# B&R Automation Studio project Panasonic_LinkaPowerCP2_A2021055 (part 34)

#### Main.st - Init, cyclic, exit code
```iecst
PROGRAM _INIT
	(* Insert code here *)

END_PROGRAM

PROGRAM _CYCLIC

	//**********************************************************IO modul Wedmuller**********************************************************************//
	//************Karta AB 4.2 8DI**************//
	P4_Etiketovacka.IN.NapajanieTlaciarne_OK := P4_Pracovisko.COM_Weidmuller.AB4_2_8DI.0;
	P4_Vytah.IN.StavRiadeniaDopravVytahu_READY := P4_Pracovisko.COM_Weidmuller.AB4_2_8DI.1;
	P4_Dopravniky.IN.StavRiadPredDopravBunky_READY := P4_Pracovisko.COM_Weidmuller.AB4_2_8DI.2;
	P4_Dopravniky.IN.StavRiadeniaPriecnDoprav_READY := P4_Pracovisko.COM_Weidmuller.AB4_2_8DI.3;
	P4_Dopravniky.IN.StavRiadZadnDopravBunky_READY := P4_Pracovisko.COM_Weidmuller.AB4_2_8DI.4;
	P4_Dopravniky.IN.StavRiadeniaVratnehoDoprav_READY := P4_Pracovisko.COM_Weidmuller.AB4_2_8DI.5;
	P4_Vytah.IN.TeplotaMotoraDopravVytahu_OK := P4_Pracovisko.COM_Weidmuller.AB4_2_8DI.6;
	P4_Dopravniky.IN.TeplotaMotoraPredDopravBunky_OK := P4_Pracovisko.COM_Weidmuller.AB4_2_8DI.7;

	//************Karta AB 4.3 8DI**************//
	P4_Dopravniky.IN.TeplotaMotoraPriecnDoprav_OK := P4_Pracovisko.COM_Weidmuller.AB4_3_8DI.0;
	P4_Dopravniky.IN.TeplotaMotoraZadnDopravBunky_OK := P4_Pracovisko.COM_Weidmuller.AB4_3_8DI.1;
	P4_Dopravniky.IN.TeplotaMotoraVratnehoDoprav_OK :=  P4_Pracovisko.COM_Weidmuller.AB4_3_8DI.2;
	P4_Pracovisko.COM_Weidmuller.AB4_3_8DI.3;
	P4_Pracovisko.COM_Weidmuller.AB4_3_8DI.4;
	P4_Pracovisko.COM_Weidmuller.AB4_3_8DI.5;
	Safety.IN.Linka_SV_ZonaCS := P4_Pracovisko.COM_Weidmuller.AB4_3_8DI.6;
	Safety.IN.P4_SV_ZonaBunky := P4_Pracovisko.COM_Weidmuller.AB4_3_8DI.7;

	//************Karta AB 4.4 8DI**************//
	Safety.IN.P4_SV_ZonaVytahu := P4_Pracovisko.COM_Weidmuller.AB4_4_8DI.0;
	Safety.IN.P4_SV_PrivodVzduchu_CH1 := P4_Pracovisko.COM_Weidmuller.AB4_4_8DI.1;
	Safety.IN.P4_SV_PrivodVzduchu_CH2 := P4_Pracovisko.COM_Weidmuller.AB4_4_8DI.2;
	P4_Pracovisko.IN.TlakVzduchu_OK := P4_Pracovisko.COM_Weidmuller.AB4_4_8DI.3;
	P4_Pracovisko.COM_Weidmuller.AB4_4_8DI.4;
	P4_Pracovisko.COM_Weidmuller.AB4_4_8DI.5;
	P4_Pracovisko.COM_Weidmuller.AB4_4_8DI.6;
	P4_Pracovisko.COM_Weidmuller.AB4_4_8DI.7;

	//************Karta AB 4.5 8DO**************//
	P4_Pracovisko.COM_Weidmuller.AB4_5_8DO.0 := P4_Pracovisko.OUT.Majak_ZeleneSvetlo_ON;
	P4_Pracovisko.COM_Weidmuller.AB4_5_8DO.1 := P4_Pracovisko.OUT.Majak_OranzoveSvetlo_ON;
	P4_Pracovisko.COM_Weidmuller.AB4_5_8DO.2 := P4_Pracovisko.OUT.Majak_CerveneSvetlo_ON;
	P4_Pracovisko.COM_Weidmuller.AB4_5_8DO.3 := P4_Pracovisko.OUT.Majak_Hukacka_ON;
	P4_Pracovisko.COM_Weidmuller.AB4_5_8DO.4;
	P4_Pracovisko.COM_Weidmuller.AB4_5_8DO.5;
	P4_Pracovisko.COM_Weidmuller.AB4_5_8DO.6 := P4_Vytah.OUT.OsvetlenieVytahu_ON;
	P4_Pracovisko.COM_Weidmuller.AB4_5_8DO.7 := P4_Pracovisko.OUT.OsvetlenieBunky_ON;

	//************Karta AB 4.6 8DO**************//
	P4_Pracovisko.COM_Weidmuller.AB4_6_8DO.0 := P4_Pracovisko.OUT.Osvetlenie_CAM15_ON;
	P4_Pracovisko.COM_Weidmuller.AB4_6_8DO.1 := P4_Vytah.OUT.DopravnikChod_VZAD;
	P4_Pracovisko.COM_Weidmuller.AB4_6_8DO.2 := P4_Vytah.OUT.DopravnikChod_VPRED;
	P4_Pracovisko.COM_Weidmuller.AB4_6_8DO.3 := P4_Dopravniky.OUT.PrednyDopravnikBunky_ON;
	P4_Pracovisko.COM_Weidmuller.AB4_6_8DO.4 := P4_Dopravniky.OUT.PriecnyDopravnik_VPRED;
	P4_Pracovisko.COM_Weidmuller.AB4_6_8DO.5 := P4_Dopravniky.OUT.ZadnyDopravnikBunky_ON;
	P4_Pracovisko.COM_Weidmuller.AB4_6_8DO.6 := P4_Dopravniky.OUT.VratnyDopravnik_ON;
	P4_Pracovisko.COM_Weidmuller.AB4_6_8DO.7 := Safety.OUT.Linka_ResetCS;

	//************Karta AB 4.8 8DO**************//
	P4_Pracovisko.COM_Weidmuller.AB4_8_8DO.0:= Safety.OUT.P4_ResetZonyBunky;
	P4_Pracovisko.COM_Weidmuller.AB4_8_8DO.1:= Safety.OUT.P4_ResetZonyVytahu;
	P4_Pracovisko.COM_Weidmuller.AB4_8_8DO.2;
	P4_Pracovisko.COM_Weidmuller.AB4_8_8DO.3;
	P4_Pracovisko.COM_Weidmuller.AB4_8_8DO.4;
	P4_Pracovisko.COM_Weidmuller.AB4_8_8DO.5;
	P4_Pracovisko.COM_Weidmuller.AB4_8_8DO.6;
	P4_Pracovisko.COM_Weidmuller.AB4_8_8DO.7;

	//**************************************************************IO modul Festo**********************************************************************************//

	//**********Modul DM 4.1 4DI4DO**************//
	//Inputs//
	P4_Pracovisko.IN.PredneDvere_PritomnostAdaptera := P4_Pracovisko.COM_Festo.DM4_1_4DI[0];
	P4_Pracovisko.IN.ZadneDvere_PritomnostAdaptera := P4_Pracovisko.COM_Festo.DM4_1_4DI[1];
	P4_ZdvizkaZaFunkcTestA.IN.TlmicPaletky_ZASUNUTY := P4_Pracovisko.COM_Festo.DM4_1_4DI[2];
	P4_Vytah.IN.PrechodDopravnika := P4_Pracovisko.COM_Festo.DM4_1_4DI[3];

	//Outputs//
	P4_Pracovisko.COM_Festo.DM4_1_4DO[0] := P4_Pracovisko.OUT.PredneDvere_ZAMKNI;
	P4_Pracovisko.COM_Festo.DM4_1_4DO[1] := P4_Pracovisko.OUT.ZadneDvere_ZAMKNI;
	P4_Pracovisko.COM_Festo.DM4_1_4DO[2];
	P4_Pracovisko.COM_Festo.DM4_1_4DO[3];

	//***********Modul DI 4.1 8DI****************//
	P4_FunkcnyTestA.IN.TypSpodnychKontaktov_5F_5H:= P4_Pracovisko.COM_Festo.DI4_1_8DI[0];
	P4_FunkcnyTestA.IN.TypSpodnychKontaktov_4F:= P4_Pracovisko.COM_Festo.DI4_1_8DI[1];
	P4_FunkcnyTestB.IN.TypSpodnychKontaktov_5F_5H:= P4_Pracovisko.COM_Festo.DI4_1_8DI[2];
	P4_FunkcnyTestB.IN.TypSpodnychKontaktov_4F:= P4_Pracovisko.COM_Festo.DI4_1_8DI[3];
	P4_Etiketovacka.IN.Centrovanie_ZASUNUTE := P4_Pracovisko.COM_Festo.DI4_1_8DI[4];
	P4_Etiketovacka.IN.Centrovanie_VYSUNUTE := P4_Pracovisko.COM_Festo.DI4_1_8DI[5];
	P4_SpodnyStoper.IN.ZaplnenieDopravnika := P4_Pracovisko.COM_Festo.DI4_1_8DI[6];
	P4_SpodnyStoper.IN.PritomnostPaletky := P4_Pracovisko.COM_Festo.DI4_1_8DI[7];

	//***********Modul DI 4.2 8DI****************//
	P4_Etiketovacka.IN.Aplikator_OtocenyVPRED := P4_Pracovisko.COM_Festo.DI4_2_8DI[0];
	P4_Etiketovacka.IN.Aplikator_OtocenyVZAD := P4_Pracovisko.COM_Festo.DI4_2_8DI[1];
	P4_Etiketovacka.IN.Aplikator_ZASUNUTY := P4_Pracovisko.COM_Festo.DI4_2_8DI[2];
	P4_Etiketovacka.IN.Aplikator_VYSUNUTY := P4_Pracovisko.COM_Festo.DI4_2_8DI[3];
	P4_Etiketovacka.IN.PritlakPowerCP_ZASUNUTY := P4_Pracovisko.COM_Festo.DI4_2_8DI[4];
	P4_Etiketovacka.IN.PritlakPowerCP_VYSUNUTY_45F := P4_Pracovisko.COM_Festo.DI4_2_8DI[5];
	P4_Etiketovacka.IN.PrisavanieEtikety_Vakum_OK := P4_Pracovisko.COM_Festo.DI4_2_8DI[6];
	P4_Etiketovacka.IN.PritlakPowerCP_VYSUNUTY_5H := P4_Pracovisko.COM_Festo.DI4_2_8DI[7];

	//***********Modul DI 4.3 8DI****************//
	P4_FunkcnyTestA.IN.HorneKontakty_VYSUNUTE := P4_Pracovisko.COM_Festo.DI4_3_8DI[0];
	P4_FunkcnyTestA.IN.HorneKontakty_ZASUNUTE := P4_Pracovisko.COM_Festo.DI4_3_8DI[1];
	P4_FunkcnyTestA.IN.Centrovanie_ZASUNUTE := P4_Pracovisko.COM_Festo.DI4_3_8DI[2];
	P4_FunkcnyTestA.IN.Centrovanie_VYSUNUTE := P4_Pracovisko.COM_Festo.DI4_3_8DI[3];
	P4_FunkcnyTestA.IN.SpodneKontakty_ZASUNUTE := P4_Pracovisko.COM_Festo.DI4_3_8DI[4];
	P4_FunkcnyTestA.IN.SpodneKontakty_VYSUNUTE := P4_Pracovisko.COM_Festo.DI4_3_8DI[5];
	P4_Pracovisko.COM_Festo.DI4_3_8DI[6];
	P4_Pracovisko.COM_Festo.DI4_3_8DI[7];

	//***********Modul DI 4.4 8DI****************//
	P4_FunkcnyTestB.IN.HorneKontakty_VYSUNUTE := P4_Pracovisko.COM_Festo.DI4_4_8DI[0];
	P4_FunkcnyTestB.IN.HorneKontakty_ZASUNUTE := P4_Pracovisko.COM_Festo.DI4_4_8DI[1];
	P4_FunkcnyTestB.IN.Centrovanie_ZASUNUTE := P4_Pracovisko.COM_Festo.DI4_4_8DI[2];
	P4_FunkcnyTestB.IN.Centrovanie_VYSUNUTE := P4_Pracovisko.COM_Festo.DI4_4_8DI[3];
	P4_FunkcnyTestB.IN.SpodneKontakty_ZASUNUTE := P4_Pracovisko.COM_Festo.DI4_4_8DI[4];
	P4_FunkcnyTestB.IN.SpodneKontakty_VYSUNUTE := P4_Pracovisko.COM_Festo.DI4_4_8DI[5];
	P4_Pracovisko.COM_Festo.DI4_4_8DI[6];
	P4_Pracovisko.COM_Festo.DI4_4_8DI[7];

	//***********Modul DI 4.5 8DI****************//
	P4_ZdvizkaZaFunkcTestA.IN.Zdvizka_HornaPoloha := P4_Pracovisko.COM_Festo.DI4_5_8DI[0];
	P4_ZdvizkaZaFunkcTestA.IN.Zdvizka_SpodnaPoloha := P4_Pracovisko.COM_Festo.DI4_5_8DI[1];
	P4_ZdvizkaZaFunkcTestA.IN.PoziciaPaletky_OK := P4_Pracovisko.COM_Festo.DI4_5_8DI[2];
	P4_ZdvizkaZaFunkcTestA.IN.Zdvizka_StrednaPoloha := P4_Pracovisko.COM_Festo.DI4_5_8DI[3];
	P4_ZdvizkaZaFunkcTestB.IN.PritomnostPaletky := P4_Pracovisko.COM_Festo.DI4_5_8DI[4];
	P4_ZdvizkaZaFunkcTestA.IN.PritomnostPaletky := P4_Pracovisko.COM_Festo.DI4_5_8DI[5];
	P4_ZdvizkaZaFunkcTestB.IN.Zdvizka_StrednaPoloha := P4_Pracovisko.COM_Festo.DI4_5_8DI[6];
	P4_ZdvizkaZaFunkcTestB.IN.Zdvizka_HornaPoloha := P4_Pracovisko.COM_Festo.DI4_5_8DI[7];

	//********Modul DS 4.1 IO link Port 0 - RFID snímač paletky funkčný test A**************//
	//Inputs//
	P4_FunkcnyTestA.RFID_hlava.Mapping_IN[0]:= P4_Pracovisko.COM_Festo.DS4_1_Port0_IN[0];
	P4_FunkcnyTestA.RFID_hlava.Mapping_IN[1]:= P4_Pracovisko.COM_Festo.DS4_1_Port0_IN[1];
	P4_FunkcnyTestA.RFID_hlava.Mapping_IN[2]:= P4_Pracovisko.COM_Festo.DS4_1_Port0_IN[2];
	P4_FunkcnyTestA.RFID_hlava.Mapping_IN[3]:= P4_Pracovisko.COM_Festo.DS4_1_Port0_IN[3];
	P4_FunkcnyTestA.RFID_hlava.Mapping_IN[4]:= P4_Pracovisko.COM_Festo.DS4_1_Port0_IN[4];
	P4_FunkcnyTestA.RFID_hlava.Mapping_IN[5]:= P4_Pracovisko.COM_Festo.DS4_1_Port0_IN[5];
	P4_FunkcnyTestA.RFID_hlava.Mapping_IN[6]:= P4_Pracovisko.COM_Festo.DS4_1_Port0_IN[6];
	P4_FunkcnyTestA.RFID_hlava.Mapping_IN[7]:= P4_Pracovisko.COM_Festo.DS4_1_Port0_IN[7];

	//Outputs//
	P4_Pracovisko.COM_Festo.DS4_1_Port0_OUT[0]:= P4_FunkcnyTestA.RFID_hlava.Mapping_OUT[0];
	P4_Pracovisko.COM_Festo.DS4_1_Port0_OUT[1]:= P4_FunkcnyTestA.RFID_hlava.Mapping_OUT[1];
	P4_Pracovisko.COM_Festo.DS4_1_Port0_OUT[2]:= P4_FunkcnyTestA.RFID_hlava.Mapping_OUT[2];
	P4_Pracovisko.COM_Festo.DS4_1_Port0_OUT[3]:= P4_FunkcnyTestA.RFID_hlava.Mapping_OUT[3];
	P4_Pracovisko.COM_Festo.DS4_1_Port0_OUT[4]:= P4_FunkcnyTestA.RFID_hlava.Mapping_OUT[4];
	P4_Pracovisko.COM_Festo.DS4_1_Port0_OUT[5]:= P4_FunkcnyTestA.RFID_hlava.Mapping_OUT[5];
	P4_Pracovisko.COM_Festo.DS4_1_Port0_OUT[6]:= P4_FunkcnyTestA.RFID_hlava.Mapping_OUT[6];
	P4_Pracovisko.COM_Festo.DS4_1_Port0_OUT[7]:= P4_FunkcnyTestA.RFID_hlava.Mapping_OUT[7];

	//********Modul DS 4.1 IO link Port 1 - RFID snímač paletky funkčný test B**************//
	//Inputs//
	P4_FunkcnyTestB.RFID_hlava.Mapping_IN[0]:= P4_Pracovisko.COM_Festo.DS4_1_Port1_IN[0];
	P4_FunkcnyTestB.RFID_hlava.Mapping_IN[1]:= P4_Pracovisko.COM_Festo.DS4_1_Port1_IN[1];
	P4_FunkcnyTestB.RFID_hlava.Mapping_IN[2]:= P4_Pracovisko.COM_Festo.DS4_1_Port1_IN[2];
	P4_FunkcnyTestB.RFID_hlava.Mapping_IN[3]:= P4_Pracovisko.COM_Festo.DS4_1_Port1_IN[3];
	P4_FunkcnyTestB.RFID_hlava.Mapping_IN[4]:= P4_Pracovisko.COM_Festo.DS4_1_Port1_IN[4];
	P4_FunkcnyTestB.RFID_hlava.Mapping_IN[5]:= P4_Pracovisko.COM_Festo.DS4_1_Port1_IN[5];
	P4_FunkcnyTestB.RFID_hlava.Mapping_IN[6]:= P4_Pracovisko.COM_Festo.DS4_1_Port1_IN[6];
	P4_FunkcnyTestB.RFID_hlava.Mapping_IN[7]:= P4_Pracovisko.COM_Festo.DS4_1_Port1_IN[7];

	//Outputs//
	P4_Pracovisko.COM_Festo.DS4_1_Port1_OUT[0]:= P4_FunkcnyTestB.RFID_hlava.Mapping_OUT[0];
	P4_Pracovisko.COM_Festo.DS4_1_Port1_OUT[1]:= P4_FunkcnyTestB.RFID_hlava.Mapping_OUT[1];
	P4_Pracovisko.COM_Festo.DS4_1_Port1_OUT[2]:= P4_FunkcnyTestB.RFID_hlava.Mapping_OUT[2];
	P4_Pracovisko.COM_Festo.DS4_1_Port1_OUT[3]:= P4_FunkcnyTestB.RFID_hlava.Mapping_OUT[3];
	P4_Pracovisko.COM_Festo.DS4_1_Port1_OUT[4]:= P4_FunkcnyTestB.RFID_hlava.Mapping_OUT[4];
	P4_Pracovisko.COM_Festo.DS4_1_Port1_OUT[5]:= P4_FunkcnyTestB.RFID_hlava.Mapping_OUT[5];
	P4_Pracovisko.COM_Festo.DS4_1_Port1_OUT[6]:= P4_FunkcnyTestB.RFID_hlava.Mapping_OUT[6];
	P4_Pracovisko.COM_Festo.DS4_1_Port1_OUT[7]:= P4_FunkcnyTestB.RFID_hlava.Mapping_OUT[7];

	//********Modul DS 4.1 IO link Port 2 - RFID snímač paletky etiketovanie**************//
	//Inputs//
	P4_Etiketovacka.RFID_hlava.Mapping_IN[0]:= P4_Pracovisko.COM_Festo.DS4_1_Port2_IN[0];
	P4_Etiketovacka.RFID_hlava.Mapping_IN[1]:= P4_Pracovisko.COM_Festo.DS4_1_Port2_IN[1];
	P4_Etiketovacka.RFID_hlava.Mapping_IN[2]:= P4_Pracovisko.COM_Festo.DS4_1_Port2_IN[2];
	P4_Etiketovacka.RFID_hlava.Mapping_IN[3]:= P4_Pracovisko.COM_Festo.DS4_1_Port2_IN[3];
	P4_Etiketovacka.RFID_hlava.Mapping_IN[4]:= P4_Pracovisko.COM_Festo.DS4_1_Port2_IN[4];
	P4_Etiketovacka.RFID_hlava.Mapping_IN[5]:= P4_Pracovisko.COM_Festo.DS4_1_Port2_IN[5];
	P4_Etiketovacka.RFID_hlava.Mapping_IN[6]:= P4_Pracovisko.COM_Festo.DS4_1_Port2_IN[6];
	P4_Etiketovacka.RFID_hlava.Mapping_IN[7]:= P4_Pracovisko.COM_Festo.DS4_1_Port2_IN[7];

	//Outputs//
	P4_Pracovisko.COM_Festo.DS4_1_Port2_OUT[0]:= P4_Etiketovacka.RFID_hlava.Mapping_OUT[0];
	P4_Pracovisko.COM_Festo.DS4_1_Port2_OUT[1]:= P4_Etiketovacka.RFID_hlava.Mapping_OUT[1];
	P4_Pracovisko.COM_Festo.DS4_1_Port2_OUT[2]:= P4_Etiketovacka.RFID_hlava.Mapping_OUT[2];
	P4_Pracovisko.COM_Festo.DS4_1_Port2_OUT[3]:= P4_Etiketovacka.RFID_hlava.Mapping_OUT[3];
	P4_Pracovisko.COM_Festo.DS4_1_Port2_OUT[4]:= P4_Etiketovacka.RFID_hlava.Mapping_OUT[4];
	P4_Pracovisko.COM_Festo.DS4_1_Port2_OUT[5]:= P4_Etiketovacka.RFID_hlava.Mapping_OUT[5];
	P4_Pracovisko.COM_Festo.DS4_1_Port2_OUT[6]:= P4_Etiketovacka.RFID_hlava.Mapping_OUT[6];
	P4_Pracovisko.COM_Festo.DS4_1_Port2_OUT[7]:= P4_Etiketovacka.RFID_hlava.Mapping_OUT[7];

	//*************Modul DS 4.2 IO link Port 0 - Banner*********************//
	//Inputs//
	P4_Vytah.Banner.Mapping_IN[0]:= P4_Pracovisko.COM_Festo.DS4_2_Port0_IN[0];
	P4_Vytah.Banner.Mapping_IN[1]:= P4_Pracovisko.COM_Festo.DS4_2_Port0_IN[1];
	P4_Vytah.Banner.Mapping_IN[2]:= P4_Pracovisko.COM_Festo.DS4_2_Port0_IN[2];
	P4_Vytah.Banner.Mapping_IN[3]:= P4_Pracovisko.COM_Festo.DS4_2_Port0_IN[3];
	P4_Vytah.Banner.Mapping_IN[4]:= P4_Pracovisko.COM_Festo.DS4_2_Port0_IN[4];
	P4_Vytah.Banner.Mapping_IN[5]:= P4_Pracovisko.COM_Festo.DS4_2_Port0_IN[5];
	P4_Vytah.Banner.Mapping_IN[6]:= P4_Pracovisko.COM_Festo.DS4_2_Port0_IN[6];
	P4_Vytah.Banner.Mapping_IN[7]:= P4_Pracovisko.COM_Festo.DS4_2_Port0_IN[7];
	P4_Vytah.Banner.Mapping_IN[8]:= P4_Pracovisko.COM_Festo.DS4_2_Port0_IN[8];
	P4_Vytah.Banner.Mapping_IN[9]:= P4_Pracovisko.COM_Festo.DS4_2_Port0_IN[9];
	P4_Vytah.Banner.Mapping_IN[10]:= P4_Pracovisko.COM_Festo.DS4_2_Port0_IN[10];
	P4_Vytah.Banner.Mapping_IN[11]:= P4_Pracovisko.COM_Festo.DS4_2_Port0_IN[11];
	P4_Vytah.Banner.Mapping_IN[12]:= P4_Pracovisko.COM_Festo.DS4_2_Port0_IN[12];
	P4_Vytah.Banner.Mapping_IN[13]:= P4_Pracovisko.COM_Festo.DS4_2_Port0_IN[13];
	P4_Vytah.Banner.Mapping_IN[14]:= P4_Pracovisko.COM_Festo.DS4_2_Port0_IN[14];
	P4_Vytah.Banner.Mapping_IN[15]:= P4_Pracovisko.COM_Festo.DS4_2_Port0_IN[15];

	//Outputs//
	P4_Pracovisko.COM_Festo.DS4_2_Port0_OUT[0]:= P4_Vytah.Banner.Mapping_OUT[0];
	P4_Pracovisko.COM_Festo.DS4_2_Port0_OUT[1]:= P4_Vytah.Banner.Mapping_OUT[1];
	P4_Pracovisko.COM_Festo.DS4_2_Port0_OUT[2]:= P4_Vytah.Banner.Mapping_OUT[2];
	P4_Pracovisko.COM_Festo.DS4_2_Port0_OUT[3]:= P4_Vytah.Banner.Mapping_OUT[3];
	P4_Pracovisko.COM_Festo.DS4_2_Port0_OUT[4]:= P4_Vytah.Banner.Mapping_OUT[4];
	P4_Pracovisko.COM_Festo.DS4_2_Port0_OUT[5]:= P4_Vytah.Banner.Mapping_OUT[5];
	P4_Pracovisko.COM_Festo.DS4_2_Port0_OUT[6]:= P4_Vytah.Banner.Mapping_OUT[6];
	P4_Pracovisko.COM_Festo.DS4_2_Port0_OUT[7]:= P4_Vytah.Banner.Mapping_OUT[7];
	P4_Pracovisko.COM_Festo.DS4_2_Port0_OUT[8]:= P4_Vytah.Banner.Mapping_OUT[8];
	P4_Pracovisko.COM_Festo.DS4_2_Port0_OUT[9]:= P4_Vytah.Banner.Mapping_OUT[9];
	P4_Pracovisko.COM_Festo.DS4_2_Port0_OUT[10]:= P4_Vytah.Banner.Mapping_OUT[10];
	P4_Pracovisko.COM_Festo.DS4_2_Port0_OUT[11]:= P4_Vytah.Banner.Mapping_OUT[11];
	P4_Pracovisko.COM_Festo.DS4_2_Port0_OUT[12]:= P4_Vytah.Banner.Mapping_OUT[12];
	P4_Pracovisko.COM_Festo.DS4_2_Port0_OUT[13]:= P4_Vytah.Banner.Mapping_OUT[13];
	P4_Pracovisko.COM_Festo.DS4_2_Port0_OUT[14]:= P4_Vytah.Banner.Mapping_OUT[14];
	P4_Pracovisko.COM_Festo.DS4_2_Port0_OUT[15]:= P4_Vytah.Banner.Mapping_OUT[15];

	//********Modul DS 4.2 IO link Port 1 - RFID snímač paletky výstupný výťah**************//
	//Inputs//
	P4_Vytah.RFID_hlava.Mapping_IN[0]:= P4_Pracovisko.COM_Festo.DS4_2_Port1_IN[0];
	P4_Vytah.RFID_hlava.Mapping_IN[1]:= P4_Pracovisko.COM_Festo.DS4_2_Port1_IN[1];
	P4_Vytah.RFID_hlava.Mapping_IN[2]:= P4_Pracovisko.COM_Festo.DS4_2_Port1_IN[2];
	P4_Vytah.RFID_hlava.Mapping_IN[3]:= P4_Pracovisko.COM_Festo.DS4_2_Port1_IN[3];
	P4_Vytah.RFID_hlava.Mapping_IN[4]:= P4_Pracovisko.COM_Festo.DS4_2_Port1_IN[4];
	P4_Vytah.RFID_hlava.Mapping_IN[5]:= P4_Pracovisko.COM_Festo.DS4_2_Port1_IN[5];
	P4_Vytah.RFID_hlava.Mapping_IN[6]:= P4_Pracovisko.COM_Festo.DS4_2_Port1_IN[6];
	P4_Vytah.RFID_hlava.Mapping_IN[7]:= P4_Pracovisko.COM_Festo.DS4_2_Port1_IN[7];

	//Outputs//
	P4_Pracovisko.COM_Festo.DS4_2_Port1_OUT[0]:= P4_Vytah.RFID_hlava.Mapping_OUT[0];
	P4_Pracovisko.COM_Festo.DS4_2_Port1_OUT[1]:= P4_Vytah.RFID_hlava.Mapping_OUT[1];
	P4_Pracovisko.COM_Festo.DS4_2_Port1_OUT[2]:= P4_Vytah.RFID_hlava.Mapping_OUT[2];
	P4_Pracovisko.COM_Festo.DS4_2_Port1_OUT[3]:= P4_Vytah.RFID_hlava.Mapping_OUT[3];
	P4_Pracovisko.COM_Festo.DS4_2_Port1_OUT[4]:= P4_Vytah.RFID_hlava.Mapping_OUT[4];
	P4_Pracovisko.COM_Festo.DS4_2_Port1_OUT[5]:= P4_Vytah.RFID_hlava.Mapping_OUT[5];
	P4_Pracovisko.COM_Festo.DS4_2_Port1_OUT[6]:= P4_Vytah.RFID_hlava.Mapping_OUT[6];
	P4_Pracovisko.COM_Festo.DS4_2_Port1_OUT[7]:= P4_Vytah.RFID_hlava.Mapping_OUT[7];

	//************************************Ventilový terminál*******************************************//
	//0-7
	P4_Pracovisko.COM_VentilovyTerminal[0].0 := P4_Etiketovacka.OUT.PrisavanieEtikety_ON;
	P4_Pracovisko.COM_VentilovyTerminal[0].1 := P4_Etiketovacka.OUT.PrisavanieEtikety_OFF;
	P4_Pracovisko.COM_VentilovyTerminal[0].2 := P4_FunkcnyTestA.OUT.ZasunStoper;
	P4_Pracovisko.COM_VentilovyTerminal[0].3 := P4_FunkcnyTestB.OUT.ZasunStoper;
	P4_Pracovisko.COM_VentilovyTerminal[0].4 := P4_ZdvizkaZaFunkcTestA.OUT.Zdvizku_VYSUN;
	P4_Pracovisko.COM_VentilovyTerminal[0].5 := P4_ZdvizkaZaFunkcTestA.OUT.Zdvizku_ZASUN;
	P4_Pracovisko.COM_VentilovyTerminal[0].6 := P4_ZdvizkaZaFunkcTestA.OUT.TlmicPaletky_VYSUN;
	P4_Pracovisko.COM_VentilovyTerminal[0].7 := P4_ZdvizkaZaFunkcTestA.OUT.TlmicPaletky_ZASUN;

	//8-15
	P4_Pracovisko.COM_VentilovyTerminal[1].0 := P4_ZdvizkaZaFunkcTestB.OUT.Zdvizku_VYSUN;
	P4_Pracovisko.COM_VentilovyTerminal[1].1 := P4_Pracovisko.OUT.ZdvizkyPneuZamok_ODOMKNI;
	P4_Pracovisko.COM_VentilovyTerminal[1].2 := P4_ZdvizkaZaFunkcTestB.OUT.TlmicPaletky_VYSUN;
	P4_Pracovisko.COM_VentilovyTerminal[1].3 := P4_Etiketovacka.OUT.ZasunStoper;
	P4_Pracovisko.COM_VentilovyTerminal[1].4 := P4_SpodnyStoper.OUT.ZasunStoper;
	P4_Pracovisko.COM_VentilovyTerminal[1].5;
	P4_Pracovisko.COM_VentilovyTerminal[1].6 := P4_FunkcnyTestA.OUT.PritlakPowerCP_VYSUN;
	P4_Pracovisko.COM_VentilovyTerminal[1].7;

	//16-23
	P4_Pracovisko.COM_VentilovyTerminal[2].0 := P4_FunkcnyTestB.OUT.PritlakPowerCP_VYSUN;
	P4_Pracovisko.COM_VentilovyTerminal[2].1;
	P4_Pracovisko.COM_VentilovyTerminal[2].2 := P4_FunkcnyTestA.OUT.KontaktyTestera_VYSUN;
	P4_Pracovisko.COM_VentilovyTerminal[2].3 := P4_FunkcnyTestB.OUT.KontaktyTestera_VYSUN;
	P4_Pracovisko.COM_VentilovyTerminal[2].4 := P4_Etiketovacka.OUT.OfukEtikety_ON;
	P4_Pracovisko.COM_VentilovyTerminal[2].5;
	P4_Pracovisko.COM_VentilovyTerminal[2].6 := P4_Etiketovacka.OUT.Aplikator_OtocVPRED;
	P4_Pracovisko.COM_VentilovyTerminal[2].7 := P4_Etiketovacka.OUT.Aplikator_OtocVZAD;

	//24-31
	P4_Pracovisko.COM_VentilovyTerminal[3].0 := P4_Etiketovacka.OUT.Aplikator_VYSUN;
	P4_Pracovisko.COM_VentilovyTerminal[3].1;
	P4_Pracovisko.COM_VentilovyTerminal[3].2 := P4_Etiketovacka.OUT.PritlakPowerCP_VYSUN;
	P4_Pracovisko.COM_VentilovyTerminal[3].3;
	P4_Pracovisko.COM_VentilovyTerminal[3].4;
	P4_Pracovisko.COM_VentilovyTerminal[3].5;
	P4_Pracovisko.COM_VentilovyTerminal[3].6 := P4_FunkcnyTestA.OUT.HorneKontakty_ZASUN;
	P4_Pracovisko.COM_VentilovyTerminal[3].7 := P4_FunkcnyTestA.OUT.HorneKontakty_VYSUN;

	//32-39
	P4_Pracovisko.COM_VentilovyTerminal[4].0 := P4_FunkcnyTestA.OUT.OdpruzHornychKontaktov_VYSUN;
	P4_Pracovisko.COM_VentilovyTerminal[4].1 := P4_FunkcnyTestA.OUT.OdpruzHornychKontaktov_ZASUN;
	P4_Pracovisko.COM_VentilovyTerminal[4].2 := P4_FunkcnyTestA.OUT.Centrovanie_VYSUN;
	P4_Pracovisko.COM_VentilovyTerminal[4].3 := P4_FunkcnyTestA.OUT.Centrovanie_ZASUN;
	P4_Pracovisko.COM_VentilovyTerminal[4].4 := P4_FunkcnyTestA.OUT.SpodneKontakty_ZASUN;
	P4_Pracovisko.COM_VentilovyTerminal[4].5 := P4_FunkcnyTestA.OUT.SpodneKontakty_VYSUN;
	P4_Pracovisko.COM_VentilovyTerminal[4].6 := P4_FunkcnyTestB.OUT.HorneKontakty_ZASUN;
	P4_Pracovisko.COM_VentilovyTerminal[4].7 := P4_FunkcnyTestB.OUT.HorneKontakty_VYSUN;

	//40-47
	P4_Pracovisko.COM_VentilovyTerminal[5].0 := P4_FunkcnyTestB.OUT.OdpruzHornychKontaktov_VYSUN;
	P4_Pracovisko.COM_VentilovyTerminal[5].1 := P4_FunkcnyTestB.OUT.OdpruzHornychKontaktov_ZASUN;
	P4_Pracovisko.COM_VentilovyTerminal[5].2 := P4_FunkcnyTestB.OUT.Centrovanie_VYSUN;
	P4_Pracovisko.COM_VentilovyTerminal[5].3 := P4_FunkcnyTestB.OUT.Centrovanie_ZASUN;
	P4_Pracovisko.COM_VentilovyTerminal[5].4 := P4_FunkcnyTestB.OUT.SpodneKontakty_ZASUN;
	P4_Pracovisko.COM_VentilovyTerminal[5].5 := P4_FunkcnyTestB.OUT.SpodneKontakty_VYSUN;
	P4_Pracovisko.COM_VentilovyTerminal[5].6 := P4_Etiketovacka.OUT.Centrovanie_VYSUN;
	P4_Pracovisko.COM_VentilovyTerminal[5].7 := P4_Etiketovacka.OUT.Centrovanie_ZASUN;

	//48-55
	P4_Pracovisko.COM_VentilovyTerminal[6].0;
	P4_Pracovisko.COM_VentilovyTerminal[6].1;
	P4_Pracovisko.COM_VentilovyTerminal[6].2;
	P4_Pracovisko.COM_VentilovyTerminal[6].3;
	P4_Pracovisko.COM_VentilovyTerminal[6].4;
	P4_Pracovisko.COM_VentilovyTerminal[6].5;
	P4_Pracovisko.COM_VentilovyTerminal[6].6;
	P4_Pracovisko.COM_VentilovyTerminal[6].7;

	//Volanie knižníc//
	P4_Etiketovacka.ServoZdvihuAplikatora();
	P4_Vytah.ServoZdvihuVytahu();

END_PROGRAM

PROGRAM _EXIT
	(* Insert code here *)

END_PROGRAM
```

### Premenne.typ
```iecst
TYPE
	AirSkrutkovaciSet_typ : 	STRUCT
		CMD : AirSkrutkovaciSet_CMD_typ;
		STAV : AirSkrutkovaciSet_STAV_typ;
		IN : AirSkrutkovaciSet_IN_typ;
		OUT : AirSkrutkovaciSet_OUT_typ;
		Internal : AirSkrutkovaciSet_Internal_typ;
		Step : USINT;
	END_STRUCT;
	AirSkrutkovaciSet_CMD_typ : 	STRUCT
		ENABLE : BOOL;
		Rezim_MANUAL : BOOL;
		PodajSkrutku : BOOL;
		VysunBrzdu : BOOL;
		ResetPoruchy : BOOL;
		RR_ZapniZasobnik : BOOL;
		RR_VysunOddelovacSkrutiek : BOOL;
		RR_VysunBrzdu : BOOL;
	END_STRUCT;
	AirSkrutkovaciSet_Internal_typ : 	STRUCT
		PocetPodaniSkrutky : USINT;
		CasZaplneniaZasobnika : TON;
		CasVypnTriediacehoVzduchu : TON;
		CasVypnZasobnika : TON;
		CasPredSpustenimZasobnika : TON;
		IdleTime_200ms : TON;
		IdleTime_1500ms : TON;
		IdleTime_1s : TON;
		IdleTime_500ms : TON;
		IdleTime_100ms : TON;
		IdleTime_2s : TON;
		IdleTime_5s : TON;
		AlarmTime_5s : TON;
		AlarmTime_10s : TON;
	END_STRUCT;
	AirSkrutkovaciSet_IN_typ : 	STRUCT
		ZasobnikSkrutiekPrazdny : BOOL;
		ZaplnenieListyZasobnika : BOOL;
		PreletSnimacZaOddelovacom : BOOL;
		PreletSnimacPredBrzdou : BOOL;
		PreletSnimacPredSkrutkovackou : BOOL;
		BrzdaVYSUNUTA : BOOL; (*Pozícia podania skrutky do skrutkovačky*)
		BrzdaZASUNUTA : BOOL; (*Pozícia čakania na skrutku zo zásobníka*)
		SkrutkovackaZASUNUTA : BOOL; (*Kontrola zasunutia skrutkovačky*)
	END_STRUCT;
	AirSkrutkovaciSet_OUT_typ : 	STRUCT
		VibropohonZasobnika_RUN : BOOL;
		TriediaciVzduch_RUN : BOOL; (*Tryska nad lištou zásobníka*)
		ZhadzovaciVzduch_RUN : BOOL; (*Tryska pred lištou zásobníka*)
		NastrelSkrutkuDoBrzdy : BOOL;
		NastrelSkrutkuDoSkrutkovacky : BOOL;
		OdsavanieBrzdy_RUN : BOOL; (*Odsávanie nečistôt z brzdy*)
		OddelovacSkrutiek_VYSUN : BOOL; (*Podanie skrutky do hadice*)
		Brzdu_VYSUN : BOOL; (*Podanie skrutky do skrutkovačky*)
		Brzdu_ZASUN : BOOL; (*Presun brzdy na pozíciu čakania skrutky zo zásobníka*)
	END_STRUCT;
	AirSkrutkovaciSet_STAV_typ : 	STRUCT
		SkrutkaPripravena : BOOL;
		ERROR : BOOL;
		PopisPoruchy : STRING[100];
		PodanieSkrutky_BUSY : BOOL;
		SkrutkovaciSet_READY : BOOL;
	END_STRUCT;
END_TYPE
```

### Variables.var
```iecst
VAR
	SkrutkSet_K30 : AirSkrutkovaciSet_typ := (0);
END_VAR
```

### Program Logical/Program/TestSkrutkSetu/Program (IEC)

#### Main.st - Init, cyclic, exit code
```iecst
PROGRAM _INIT
	(* Insert code here *)

END_PROGRAM

PROGRAM _CYCLIC

	//********************************Zrušenie príznaku skrutka pripravena**********************************************************//
	IF SkrutkSet_K30.STAV.SkrutkaPripravena AND NOT SkrutkSet_K30.IN.SkrutkovackaZASUNUTA THEN
		SkrutkSet_K30.STAV.SkrutkaPripravena:= FALSE;
	END_IF

	//*******************************Ovládanie zhadzovacieho vzduchu pred lištou zásobníka******************************************//
	SkrutkSet_K30.Internal.CasZaplneniaZasobnika.IN:= SkrutkSet_K30.IN.ZaplnenieListyZasobnika AND SkrutkSet_K30.OUT.VibropohonZasobnika_RUN;

	IF SkrutkSet_K30.Internal.CasZaplneniaZasobnika.Q THEN
		SkrutkSet_K30.OUT.ZhadzovaciVzduch_RUN:= TRUE;
	ELSIF NOT SkrutkSet_K30.OUT.VibropohonZasobnika_RUN THEN
		SkrutkSet_K30.OUT.ZhadzovaciVzduch_RUN:= FALSE;
	ELSE
		SkrutkSet_K30.OUT.ZhadzovaciVzduch_RUN:= FALSE;
	END_IF

	SkrutkSet_K30.Internal.CasZaplneniaZasobnika.PT:= T#3s;
	SkrutkSet_K30.Internal.CasZaplneniaZasobnika();

	//******************************Vypnutie triediaceho vzduchu nad lištou zásobníka************************************************//
	SkrutkSet_K30.Internal.CasVypnTriediacehoVzduchu.IN:= SkrutkSet_K30.OUT.TriediaciVzduch_RUN AND NOT SkrutkSet_K30.OUT.VibropohonZasobnika_RUN;
	IF SkrutkSet_K30.Internal.CasVypnTriediacehoVzduchu.Q THEN
		SkrutkSet_K30.OUT.TriediaciVzduch_RUN:= FALSE;
	END_IF

	SkrutkSet_K30.Internal.CasVypnTriediacehoVzduchu.PT:= T#1s;
	SkrutkSet_K30.Internal.CasVypnTriediacehoVzduchu();

	//********************************Vypnutie zásobníka**************************************************************//
	SkrutkSet_K30.Internal.CasVypnZasobnika.IN:= SkrutkSet_K30.IN.ZaplnenieListyZasobnika AND SkrutkSet_K30.OUT.VibropohonZasobnika_RUN AND NOT SkrutkSet_K30.CMD.RR_ZapniZasobnik;

	IF SkrutkSet_K30.Internal.CasVypnZasobnika.Q THEN
		SkrutkSet_K30.OUT.VibropohonZasobnika_RUN:= FALSE;
	END_IF

	SkrutkSet_K30.Internal.CasVypnZasobnika.PT:= T#3s;
	SkrutkSet_K30.Internal.CasVypnZasobnika();

	//*******************************Zapnutie zásobníka keď je prázdna lišta zásobníka*****************//
	IF SkrutkSet_K30.CMD.ENABLE AND NOT SkrutkSet_K30.STAV.ERROR AND NOT SkrutkSet_K30.IN.ZaplnenieListyZasobnika AND NOT SkrutkSet_K30.OUT.VibropohonZasobnika_RUN AND NOT SkrutkSet_K30.OUT.OddelovacSkrutiek_VYSUN THEN
		SkrutkSet_K30.OUT.VibropohonZasobnika_RUN:= TRUE;
	END_IF

	//***************************Ručný režim**************************************************//
	//Ovládanie zásobníka//
	IF SkrutkSet_K30.CMD.Rezim_MANUAL AND NOT SkrutkSet_K30.STAV.PodanieSkrutky_BUSY THEN
		IF SkrutkSet_K30.Internal.CasPredSpustenimZasobnika.Q THEN
			SkrutkSet_K30.OUT.VibropohonZasobnika_RUN:= TRUE;
		ELSE
			SkrutkSet_K30.OUT.VibropohonZasobnika_RUN:= FALSE;
		END_IF
	END_IF

	SkrutkSet_K30.Internal.CasPredSpustenimZasobnika.IN:= SkrutkSet_K30.CMD.Rezim_MANUAL AND SkrutkSet_K30.CMD.RR_ZapniZasobnik;
	SkrutkSet_K30.Internal.CasPredSpustenimZasobnika.PT:= T#1s;
	SkrutkSet_K30.Internal.CasPredSpustenimZasobnika();

	//Ovládanie brzdy//
	IF SkrutkSet_K30.CMD.Rezim_MANUAL AND NOT SkrutkSet_K30.STAV.PodanieSkrutky_BUSY THEN
		IF SkrutkSet_K30.CMD.RR_VysunBrzdu THEN
			SkrutkSet_K30.OUT.Brzdu_VYSUN:= TRUE;
			SkrutkSet_K30.OUT.Brzdu_ZASUN:= FALSE;
		ELSE
			SkrutkSet_K30.OUT.Brzdu_VYSUN:= FALSE;
			SkrutkSet_K30.OUT.Brzdu_ZASUN:= TRUE;
		END_IF
	END_IF

	//Ovládanie oddelovača skrutiek//
	IF SkrutkSet_K30.CMD.Rezim_MANUAL AND NOT SkrutkSet_K30.STAV.PodanieSkrutky_BUSY THEN
		IF SkrutkSet_K30.CMD.RR_VysunOddelovacSkrutiek THEN
			SkrutkSet_K30.OUT.OddelovacSkrutiek_VYSUN:= TRUE;
		ELSE
			SkrutkSet_K30.OUT.OddelovacSkrutiek_VYSUN:= FALSE;
		END_IF
	END_IF

	//***********************************Enable knižnice***************************************//
	IF NOT SkrutkSet_K30.CMD.ENABLE AND SkrutkSet_K30.Step <> 0 THEN
		SkrutkSet_K30.OUT.VibropohonZasobnika_RUN:= FALSE;
		SkrutkSet_K30.Step:= 0;
	END_IF

	//**********************************Reset poruchy*****************************************//
	IF SkrutkSet_K30.CMD.ResetPoruchy OR NOT SkrutkSet_K30.CMD.ENABLE THEN
		SkrutkSet_K30.STAV.ERROR:= FALSE;
		SkrutkSet_K30.STAV.PopisPoruchy:= '';
		SkrutkSet_K30.CMD.ResetPoruchy:= FALSE;
	END_IF

	CASE SkrutkSet_K30.Step OF

		0: //Nulovanie//
			SkrutkSet_K30.Internal.IdleTime_200ms.IN:= FALSE;
			SkrutkSet_K30.Internal.IdleTime_100ms.IN:= FALSE;
			SkrutkSet_K30.Internal.IdleTime_500ms.IN:= FALSE;
			SkrutkSet_K30.Internal.IdleTime_1s.IN:= FALSE;
			SkrutkSet_K30.Internal.IdleTime_2s.IN:= FALSE;
			SkrutkSet_K30.Internal.IdleTime_5s.IN:= FALSE;
			SkrutkSet_K30.Internal.IdleTime_1500ms.IN:= FALSE;
			SkrutkSet_K30.Internal.AlarmTime_5s.IN:= FALSE;
			SkrutkSet_K30.Internal.AlarmTime_10s.IN:= FALSE;
			SkrutkSet_K30.Internal.PocetPodaniSkrutky:= 0;
			SkrutkSet_K30.OUT.Brzdu_VYSUN:= FALSE;
			SkrutkSet_K30.OUT.Brzdu_ZASUN:= TRUE;
			SkrutkSet_K30.OUT.OddelovacSkrutiek_VYSUN:= FALSE;
			SkrutkSet_K30.OUT.NastrelSkrutkuDoBrzdy:= FALSE;
			SkrutkSet_K30.OUT.NastrelSkrutkuDoSkrutkovacky:= FALSE;
			SkrutkSet_K30.OUT.OdsavanieBrzdy_RUN:= FALSE;
			SkrutkSet_K30.CMD.Rezim_MANUAL:= FALSE;
			SkrutkSet_K30.CMD.PodajSkrutku:= FALSE;
			SkrutkSet_K30.CMD.VysunBrzdu:= FALSE;
			SkrutkSet_K30.CMD.RR_ZapniZasobnik:= FALSE;
			SkrutkSet_K30.CMD.RR_VysunBrzdu:= FALSE;
			SkrutkSet_K30.CMD.RR_VysunOddelovacSkrutiek:= FALSE;
			SkrutkSet_K30.STAV.PodanieSkrutky_BUSY:= FALSE;
			SkrutkSet_K30.STAV.SkrutkovaciSet_READY:= FALSE;

			IF SkrutkSet_K30.CMD.ENABLE AND NOT SkrutkSet_K30.STAV.ERROR THEN
				SkrutkSet_K30.Step:= 1;
			END_IF

		1: //Čakam na spustenie//
			SkrutkSet_K30.STAV.SkrutkovaciSet_READY:= TRUE;
			IF SkrutkSet_K30.CMD.PodajSkrutku THEN
				SkrutkSet_K30.STAV.SkrutkovaciSet_READY:= FALSE;
				SkrutkSet_K30.STAV.PodanieSkrutky_BUSY:= TRUE;
				SkrutkSet_K30.Step:= 10;
			ELSIF SkrutkSet_K30.CMD.VysunBrzdu THEN
				SkrutkSet_K30.STAV.SkrutkovaciSet_READY:= FALSE;
				SkrutkSet_K30.STAV.PodanieSkrutky_BUSY:= TRUE;
				SkrutkSet_K30.Step:= 30;
			END_IF

		10: //Vysunutie brzdy pre kontrolu skrutky v brzde, kontrola preletu skrutky cez preletovy snimac pred skrutkovackou//
			SkrutkSet_K30.OUT.Brzdu_ZASUN:= FALSE;
			SkrutkSet_K30.OUT.Brzdu_VYSUN:= TRUE;
			SkrutkSet_K30.Internal.AlarmTime_5s.IN:= NOT SkrutkSet_K30.IN.BrzdaVYSUNUTA;

			IF SkrutkSet_K30.IN.BrzdaVYSUNUTA THEN
				SkrutkSet_K30.OUT.NastrelSkrutkuDoSkrutkovacky:= TRUE;
				SkrutkSet_K30.Internal.IdleTime_2s.IN:= TRUE;
			END_IF

			IF SkrutkSet_K30.IN.PreletSnimacPredSkrutkovackou THEN
				SkrutkSet_K30.Internal.AlarmTime_5s.IN:= FALSE;
				SkrutkSet_K30.Internal.IdleTime_2s.IN:= FALSE;
				SkrutkSet_K30.STAV.SkrutkaPripravena:= TRUE;
				SkrutkSet_K30.Step:= 13;
			ELSIF SkrutkSet_K30.Internal.IdleTime_2s.Q THEN
				SkrutkSet_K30.Internal.AlarmTime_5s.IN:= FALSE;
				SkrutkSet_K30.Internal.IdleTime_2s.IN:= FALSE;
				SkrutkSet_K30.Step:= 13;
			ELSIF SkrutkSet_K30.Internal.AlarmTime_5s.Q THEN
				SkrutkSet_K30.STAV.ERROR:= TRUE;
				SkrutkSet_K30.STAV.PopisPoruchy:= 'Porucha vysunutia brzdy';
				SkrutkSet_K30.Step:= 0;
			END_IF

		13: //Vypnutie vzduchu nastrelenia skrutky do skrutkovacky a zasunutie brzdy//
			SkrutkSet_K30.OUT.NastrelSkrutkuDoSkrutkovacky:= FALSE;
			SkrutkSet_K30.OUT.Brzdu_ZASUN:= TRUE;
			SkrutkSet_K30.OUT.Brzdu_VYSUN:= FALSE;
			SkrutkSet_K30.Internal.AlarmTime_5s.IN:= NOT SkrutkSet_K30.IN.BrzdaZASUNUTA;

			IF SkrutkSet_K30.IN.BrzdaZASUNUTA THEN
				SkrutkSet_K30.Internal.AlarmTime_5s.IN:= FALSE;
				SkrutkSet_K30.Step:= 15;
			ELSIF SkrutkSet_K30.Internal.AlarmTime_5s.Q THEN
				SkrutkSet_K30.STAV.ERROR:= TRUE;
				SkrutkSet_K30.STAV.PopisPoruchy:= 'Porucha zasunutia brzdy';
				SkrutkSet_K30.Step:= 0;
			END_IF

		15: //Spustenie zasobnika a kontrola snimaca zaplnenia listy//
			SkrutkSet_K30.OUT.OddelovacSkrutiek_VYSUN:= FALSE;
			SkrutkSet_K30.OUT.TriediaciVzduch_RUN:= TRUE;
			SkrutkSet_K30.Internal.IdleTime_1s.IN:= SkrutkSet_K30.OUT.TriediaciVzduch_RUN;
			SkrutkSet_K30.Internal.IdleTime_1500ms.IN:= SkrutkSet_K30.IN.ZaplnenieListyZasobnika AND SkrutkSet_K30.OUT.VibropohonZasobnika_RUN;

			IF SkrutkSet_K30.Internal.IdleTime_1s.Q THEN
				SkrutkSet_K30.OUT.VibropohonZasobnika_RUN:= TRUE;
			END_IF

			IF SkrutkSet_K30.Internal.IdleTime_1500ms.Q THEN
				SkrutkSet_K30.Internal.IdleTime_1s.IN:= FALSE;
				SkrutkSet_K30.Internal.IdleTime_1500ms.IN:= FALSE;
				SkrutkSet_K30.Step:= 18;
			END_IF

		18: //Vysunutie oddelovaca skrutiek a zapnutie vzduchu nastrelenia skrutky do brzdy a zapnutie odsavania necistot
			SkrutkSet_K30.OUT.OddelovacSkrutiek_VYSUN:= TRUE;
			SkrutkSet_K30.OUT.NastrelSkrutkuDoBrzdy:= TRUE;
			SkrutkSet_K30.OUT.OdsavanieBrzdy_RUN:= TRUE;
			SkrutkSet_K30.Internal.IdleTime_2s.IN:= TRUE;

			IF SkrutkSet_K30.IN.PreletSnimacPredBrzdou THEN
				SkrutkSet_K30.Internal.IdleTime_2s.IN:= FALSE;
				SkrutkSet_K30.OUT.NastrelSkrutkuDoBrzdy:= FALSE;
				SkrutkSet_K30.OUT.OddelovacSkrutiek_VYSUN:= FALSE;
				SkrutkSet_K30.OUT.OdsavanieBrzdy_RUN:= FALSE;
				SkrutkSet_K30.Step:= 20;
			ELSIF SkrutkSet_K30.Internal.IdleTime_2s.Q THEN
				SkrutkSet_K30.Internal.IdleTime_2s.IN:= FALSE;
				SkrutkSet_K30.OUT.NastrelSkrutkuDoBrzdy:= FALSE;
				SkrutkSet_K30.OUT.OddelovacSkrutiek_VYSUN:= FALSE;
				SkrutkSet_K30.OUT.OdsavanieBrzdy_RUN:= FALSE;
				SkrutkSet_K30.Step:= 15;
			END_IF

		20: //Kontrola stavu skrutka pripravena//
			IF SkrutkSet_K30.STAV.SkrutkaPripravena THEN
				SkrutkSet_K30.Step:= 0;
			ELSE
				SkrutkSet_K30.Internal.PocetPodaniSkrutky:= SkrutkSet_K30.Internal.PocetPodaniSkrutky + 1;
				IF SkrutkSet_K30.Internal.PocetPodaniSkrutky < 4 THEN
					SkrutkSet_K30.Step:= 10;
				ELSE
					SkrutkSet_K30.STAV.ERROR:= TRUE;
					SkrutkSet_K30.STAV.PopisPoruchy:= 'Porucha nastrelenia skrutky do brzdy';
					SkrutkSet_K30.Step:= 0;
				END_IF
			END_IF

		30: //Vysunutie brzdy//
			SkrutkSet_K30.OUT.Brzdu_ZASUN:= FALSE;
			SkrutkSet_K30.OUT.Brzdu_VYSUN:= TRUE;
			SkrutkSet_K30.Internal.AlarmTime_5s.IN:= NOT SkrutkSet_K30.IN.BrzdaVYSUNUTA;

			IF NOT SkrutkSet_K30.CMD.VysunBrzdu THEN
				SkrutkSet_K30.Step:= 0;
			ELSIF SkrutkSet_K30.Internal.AlarmTime_5s.Q THEN
				SkrutkSet_K30.STAV.ERROR:= TRUE;
				SkrutkSet_K30.STAV.PopisPoruchy:= 'Porucha vysunutia brzdy';
				SkrutkSet_K30.Step:= 0;
			END_IF

	END_CASE

	//*********************************Časovače**************************************//
	SkrutkSet_K30.Internal.IdleTime_200ms.PT:= T#200ms;
	SkrutkSet_K30.Internal.IdleTime_200ms();
	SkrutkSet_K30.Internal.IdleTime_100ms.PT:= T#100ms;
	SkrutkSet_K30.Internal.IdleTime_100ms();
	SkrutkSet_K30.Internal.IdleTime_1500ms.PT:= T#1s500ms;
	SkrutkSet_K30.Internal.IdleTime_1500ms();
	SkrutkSet_K30.Internal.IdleTime_500ms.PT:= T#500ms;
	SkrutkSet_K30.Internal.IdleTime_500ms();
	SkrutkSet_K30.Internal.IdleTime_1s.PT:= T#1s;
	SkrutkSet_K30.Internal.IdleTime_1s();
	SkrutkSet_K30.Internal.IdleTime_2s.PT:= T#2s;
	SkrutkSet_K30.Internal.IdleTime_2s();
	SkrutkSet_K30.Internal.IdleTime_5s.PT:= T#5s;
	SkrutkSet_K30.Internal.IdleTime_5s();
	SkrutkSet_K30.Internal.AlarmTime_5s.PT:= T#5s;
	SkrutkSet_K30.Internal.AlarmTime_5s();
	SkrutkSet_K30.Internal.AlarmTime_10s.PT:= T#10s;
	SkrutkSet_K30.Internal.AlarmTime_10s();

END_PROGRAM

PROGRAM _EXIT
	(* Insert code here *)

END_PROGRAM
```

- Visualisation Logical/mappView (not shown)

### Program Logical/RemanentnePremenne/P1_RemanentnePremenne (IEC)

#### Main.st - Init, cyclic, exit code
```iecst
PROGRAM _INIT
	(* Insert code here *)

END_PROGRAM

PROGRAM _CYCLIC

	P1_RemPremenne;

	//Načítanie premenných pri prvom spustení//
	IF EDGEPOS(Safety.STAV.Linka_SafetyPLC_Nabehlo) THEN
		P1_NacitajPremenne:= TRUE;
	END_IF

	//Načítanie premenných z pamäte//
	IF P1_NacitajPremenne THEN
		MpRecipeXml_P1.Load:= TRUE;
		P1_NacitajPremenne:= FALSE;
	END_IF

	IF MpRecipeXml_P1.Load AND (MpRecipeXml_P1.CommandDone OR MpRecipeXml_P1.Error) THEN
		MpRecipeXml_P1.Load:= FALSE;
	END_IF

	//Konfigurácia premenných//
	MpRecipeXml_P1.MpLink:= ADR(gRemPremenneP1);  //takto sa menuje mapp komponenta v configurating view//
	MpRecipeXml_P1.Enable:= TRUE;
	MpRecipeXml_P1.Category:= ADR('PREMENNE_P1');
	MpRecipeXml_P1.DeviceName:= ADR('HDD_RemPremenneP1');  //Názov media, kde sa budú receptury ukladat//
	MpRecipeXml_P1.FileName:= ADR('RemPremenneP1'); //Názov súboru do ktorého sa receptúry uložia//
	MpRecipeXml_P1();

	MpRecipeRegPar_P1.MpLink:= ADR(gRemPremenneP1);
	MpRecipeRegPar_P1.Enable:= TRUE;
	MpRecipeRegPar_P1.Category:= ADR('PREMENNE_P1');
	MpRecipeRegPar_P1.PVName:= ADR('P1_RemPremenne'); //Názov premenné, kde je vytvorená štruktura dat premennych//
	MpRecipeRegPar_P1();

	//Uloženie premenných//
	IF P1_UlozPremenne THEN
		MpRecipeXml_P1.Save:= TRUE;
		P1_UlozPremenne:= FALSE;
	END_IF

	IF MpRecipeXml_P1.Save AND (MpRecipeXml_P1.CommandDone OR MpRecipeXml_P1.Error) THEN
		MpRecipeXml_P1.Save:= FALSE;
	END_IF

END_PROGRAM

PROGRAM _EXIT
	(* Insert code here *)

END_PROGRAM
```

#### Variables.var - Local variables
```iecst
VAR
	UISetup : MpRecipeUISetupType;
	UIConnect : MpRecipeUIConnectType := (0);
END_VAR
```

### Program Logical/RemanentnePremenne/P2_RemanentnePremenne (IEC)

#### Main.st - Init, cyclic, exit code
```iecst
PROGRAM _INIT

END_PROGRAM

PROGRAM _CYCLIC

	P2_RemPremenne;

	//Načítanie premenných pri prvom spustení//
	IF EDGEPOS(Safety.STAV.Linka_SafetyPLC_Nabehlo) THEN
		P2_NacitajPremenne:= TRUE;
	END_IF

	//Načítanie premenných z pamäte//
	IF P2_NacitajPremenne THEN
		MpRecipeXml_P2.Load:= TRUE;
		P2_NacitajPremenne:= FALSE;
	END_IF

	IF MpRecipeXml_P2.Load AND (MpRecipeXml_P2.CommandDone OR MpRecipeXml_P2.Error) THEN
		MpRecipeXml_P2.Load:= FALSE;
	END_IF

	//Konfigurácia premenných//
	MpRecipeXml_P2.MpLink:= ADR(gRemPremenneP2);  //takto sa menuje mapp komponenta v configurating view//
	MpRecipeXml_P2.Enable:= TRUE;
	MpRecipeXml_P2.Category:= ADR('PREMENNE_P2');
	MpRecipeXml_P2.DeviceName:= ADR('HDD_RemPremenneP2');  //Názov media, kde sa budú receptury ukladat//
	MpRecipeXml_P2.FileName:= ADR('RemPremenneP2'); //Názov súboru do ktorého sa receptúry uložia//
	MpRecipeXml_P2();

	MpRecipeRegPar_P2.MpLink:= ADR(gRemPremenneP2);
	MpRecipeRegPar_P2.Enable:= TRUE;
	MpRecipeRegPar_P2.Category:= ADR('PREMENNE_P2');
	MpRecipeRegPar_P2.PVName:= ADR('P2_RemPremenne'); //Názov premenné, kde je vytvorená štruktura dat premenných//
	MpRecipeRegPar_P2();

	//Uloženie premenných//
	IF P2_UlozPremenne THEN
		MpRecipeXml_P2.Save:= TRUE;
		P2_UlozPremenne:= FALSE;
	END_IF

	IF MpRecipeXml_P2.Save AND (MpRecipeXml_P2.CommandDone OR MpRecipeXml_P2.Error) THEN
		MpRecipeXml_P2.Save:= FALSE;
	END_IF

END_PROGRAM

PROGRAM _EXIT
	(* Insert code here *)

END_PROGRAM
```

#### Variables.var - Local variables
```iecst
VAR
	UISetup : MpRecipeUISetupType;
	UIConnect : MpRecipeUIConnectType := (0);
END_VAR
```

### Program Logical/RemanentnePremenne/P34_RemanentnePremenne (IEC)

#### Main.st - Init, cyclic, exit code
```iecst
PROGRAM _INIT
	(* Insert code here *)

END_PROGRAM

PROGRAM _CYCLIC

	P34_RemPremenne;
	//Načítanie premenných pri prvom spustení//
	IF EDGEPOS(Safety.STAV.Linka_SafetyPLC_Nabehlo) THEN
		P34_NacitajPremenne:= TRUE;
	END_IF

	//Načítanie premenných z pamäte//
	IF P34_NacitajPremenne THEN
		MpRecipeXml_P34.Load:= TRUE;
		P34_NacitajPremenne:= FALSE;
	END_IF

	IF MpRecipeXml_P34.Load AND (MpRecipeXml_P34.CommandDone OR MpRecipeXml_P34.Error) THEN
		MpRecipeXml_P34.Load:= FALSE;
	END_IF

	//Konfigurácia premenných//
	MpRecipeXml_P34.MpLink:= ADR(gRemPremenneP34);  //takto sa menuje mapp komponenta v configurating view//
	MpRecipeXml_P34.Enable:= TRUE;
	MpRecipeXml_P34.Category:= ADR('PREMENNE_P34');
	MpRecipeXml_P34.DeviceName:= ADR('HDD_RemPremenneP34');  //Názov media, kde sa budú receptury ukladat//
	MpRecipeXml_P34.FileName:= ADR('RemPremenneP34'); //Názov súboru do ktorého sa receptúry uložia//
	MpRecipeXml_P34();

	MpRecipeRegPar_P34.MpLink:= ADR(gRemPremenneP34);
	MpRecipeRegPar_P34.Enable:= TRUE;
	MpRecipeRegPar_P34.Category:= ADR('PREMENNE_P34');
	MpRecipeRegPar_P34.PVName:= ADR('P34_RemPremenne'); //Názov premenné, kde je vytvorená štruktura dat premennych//
	MpRecipeRegPar_P34();

	//Uloženie premenných//
	IF P34_UlozPremenne THEN
		MpRecipeXml_P34.Save:= TRUE;
		P34_UlozPremenne:= FALSE;
	END_IF

	IF MpRecipeXml_P34.Save AND (MpRecipeXml_P34.CommandDone OR MpRecipeXml_P34.Error) THEN
		MpRecipeXml_P34.Save:= FALSE;
	END_IF

END_PROGRAM

PROGRAM _EXIT
	(* Insert code here *)

END_PROGRAM
```

#### Variables.var - Local variables
```iecst
VAR
	UISetup : MpRecipeUISetupType;
	UIConnect : MpRecipeUIConnectType := (0);
END_VAR
```

### AlarmyGlobal.typ - Global data types
```iecst
TYPE
	AlarmyVizu_typ : 	STRUCT
		PotvrdAlarmy : BOOL;
		ArchivaciaAlarmov : BOOL;
		ZobrazSymbolAlarmu : USINT;
		FarbaTlacitka_Alarmy : WSTRING[80];
	END_STRUCT;
END_TYPE
```

### AlarmyGlobal.var - Global variables
```iecst
VAR
	NastalaPorucha : BOOL;
	P1_AlarmyVizu : AlarmyVizu_typ;
	P2_AlarmyVizu : AlarmyVizu_typ;
	P34_AlarmyVizu : AlarmyVizu_typ;
	P1_Alarmy : ARRAY[100..199] OF BOOL;
	P2_Alarmy : ARRAY[200..299] OF BOOL;
	P34_Alarmy : ARRAY[300..499] OF BOOL;
	MpAlarmXCore_1 : MpAlarmXCore;
	MpAlarmXHistory_1 : MpAlarmXHistory;
END_VAR
```

### Program Logical/Alarmy/P1_Alarmy (IEC)

#### Main.st - Init, cyclic, exit code
```iecst
PROGRAM _INIT
	(* Insert code here *)

END_PROGRAM

PROGRAM _CYCLIC

	//Alarmy pracoviska č.1 (100 - 199)//
	//A100 - ST1_Vytah - paletka na vystupe dopravnika vytahu !!!
	//A101 - ST1_Vytah - narusenie optickej bariery !!!
	//A102 - ST1_Vytah - porucha navezenia paletky na dopravnik vytahu !!!
	//A103 - ST1_Vytah - porucha precitania kodu paletky !!!
	//A104 - ST1_Vytah - porucha komunikacie zo serverom !!!
	//A105 - ST1_Vytah - porucha odoslania fotiek na server !!!
	//A106 - ST1_Vytah - CAM 2 porucha komunikacie FTP !!!
	//A107 - ST1_Vytah - CAM 3 porucha komunikacie FTP !!!
	//A108 - ST1_Vytah - CAM 4 porucha komunikacie FTP !!!
	//A109 - ST1_Vytah - CAM 5 porucha komunikacie FTP !!!
	//A110 - ST1_Vytah - porucha serva zdvihu vytahu !!!
	//A111 - ST2_Srobovanie - porucha vysunutia centrovacky !!!
	//A112 - ST2_Srobovanie - porucha zasunutia centrovacky !!!
	//A113 - ST2_Srobovanie - porucha precitania kodu paletky !!!
	//A114 - ST2_Srobovanie - porucha komunikacie zo serverom !!!
	//A115 - ST2_Srobovanie - porucha odoslania fotiek na server !!!
	//A116 - ST2_Srobovanie - CAM 6 porucha komunikacie FTP !!!
	//A117 - ST2_Srobovanie - porucha serva manipulatora os X !!!
	//A118 - ST2_Srobovanie - porucha serva manipulatora os Y !!!
	//A119 - ST2_Srobovanie - skrutka K30 nieje pripravena !!!
	//A120 - ST2_Srobovanie - skrutka M5 nieje pripravena !!!
    //A121 - ST2_Srobovanie - skrutka M4 nieje pripravena !!!
    //A122 - P1_Robot - porucha napajania !!!
    //A123 - P1_Robot - nieje online !!!
    //A124 - Pracovisko 1 - Porucha tlaku vzduchu !!!
    //A125 - Pracovisko 1 - Modul DI11 nieje online !!!
    //A126 - Pracovisko 1 - Modul DI12 nieje online !!!
    //A127 - Pracovisko 1 - Modul DI13 nieje online !!!
    //A128 - Pracovisko 1 - Modul DI14 nieje online !!!
    //A129 - Pracovisko 1 - Modul DM11 nieje online !!!
    //A130 - Pracovisko 1 - Modul DS11 nieje online !!!
	//A131 - Pracovisko 1 - Modul DS12 nieje online !!!
	//A132 - Pracovisko 1 - Modul SI11 nieje online !!!
	//A133 - Pracovisko 1 - Modul SI12 nieje online !!!
    //A134 - Pracovisko 1 - Ventilovy termnal VT4 nieje online !!!
    //A135 - Pracovisko 1 - Ventilovy termnal VT5 nieje online !!!
    //A136 - ST2_Srobovanie - Skrutkovacka K30 nieje online !!!
    //A137 - ST2_Srobovanie - Skrutkovacka M5 nieje online !!!
    //A138 - ST2_Srobovanie - Skrutkovacka M4 nieje online !!!
    //A139 - Pracovisko 1 - Kamery KAM2, KAM4 a KAM6 niesu online !!!
    //A140 - Pracovisko 1 - Kamera KAM3 nieje online !!!
	//A141 - Pracovisko 1 - Kamera KAM5 nieje online !!!
    //A142 - ST2_Srobovanie - Porucha vysunutia skrutkovacky K30 !!!
    //A143 - ST2_Srobovanie - Porucha vysunutia skrutkovacky M5  !!!
    //A144 - ST2_Srobovanie - Porucha vysunutia skrutkovacky M4 !!!
	//A145 - P1_Robot - porucha !!!
    //A146 - ST2_Srobovanie - Presiahnuty cas skrutkovania skrutky K30 !!!
    //A147 - ST2_Srobovanie - Presiahnuty cas skrutkovania skrutky M5 !!!
    //A148 - ST2_Srobovanie - Presiahnuty cas skrutkovania skrutky M4 !!!
    //A149 - ST2_Srobovanie - Skrutkovacka K30 nieje READY !!!
    //A150 - ST2_Srobovanie - Skrutkovacka M5 nieje READY !!!
    //A151 - ST2_Srobovanie - Skrutkovacka M4 nieje READY !!!
    //A152 - Pracovisko 1 - Prekrocena teplota motora vrchneho dopravnika !!!
    //A153 - Pracovisko 1 - Prekrocena teplota motora spodneho dopravnika !!!
    //A154 - Pracovisko 1 - Narusenie optickej bariery na vstupe !!!
    //A155 - ST1_Vytah - Prekrocena teplota motora dopravnika !!!
    //A156 - Pracovisko 1 - Bolo stlacene tlacitko CS na ovladacom paneli !!!
    //A157 - Pracovisko 1 - Bolo stlacene tlacitko CS na rozvodnej skrini !!!
    //A158 - Pracovisko 1 - Bolo stlacene tlacitko CS robota !!!
    //A159 - P1_Robot - Porucha odobratia foamov z paletky !!!
    //A160 - P1_Robot - Porucha odobratia busbarov z paletky !!!
    //A161 - ST2_Srobovanie - Porucha vyvezenia paletky zo stopra !!!
    //A162 - P1_Akumulacny stoper - Porucha vyvezenia paletky zo stopra !!!
    //A163 - P1_Spodny stoper - Porucha vyvezenia paletky zo stopra !!!
    //A164 - ST1_Vytah - Porucha komunikacie s kamerou CAM 2 !!!
    //A165 - ST1_Vytah - Porucha komunikacie s kamerou CAM 5 !!!
    //A166 - ST1_Vytah - Porucha komunikacie s kamerou CAM 4 !!!
    //A167 - ST1_Vytah - Porucha komunikacie s kamerou CAM 3 !!!
    //A168 - ST2_Srobovanie - Porucha komunikacie s kamerou CAM 6 !!!

	//******************************Configurácia alarmov**************************************//
	MpAlarmXCore_1.Enable:= TRUE;
	MpAlarmXCore_1.MpLink:= ADR(gAlarmXCore);
	MpAlarmXCore_1();

	//*****************************Configurácia histórie alarmov*****************************//

	MpAlarmXHistory_1.Enable:= TRUE;
	MpAlarmXHistory_1.MpLink:= ADR(gAlarmXHistory);
	MpAlarmXHistory_1.DeviceName:= ADR('HDD_AlarmHistory');
	MpAlarmXHistory_1();

	//****************************Archivácia alarmov na disk PLC******************************//
	IF P1_AlarmyVizu.ArchivaciaAlarmov THEN
		MpAlarmXHistory_1.Export:= TRUE;
		P1_AlarmyVizu.ArchivaciaAlarmov:= FALSE;
	ELSIF P2_AlarmyVizu.ArchivaciaAlarmov THEN
		MpAlarmXHistory_1.Export:= TRUE;
		P2_AlarmyVizu.ArchivaciaAlarmov:= FALSE;
	ELSIF P34_AlarmyVizu.ArchivaciaAlarmov THEN
		MpAlarmXHistory_1.Export:= TRUE;
		P34_AlarmyVizu.ArchivaciaAlarmov:= FALSE;
	END_IF

	IF MpAlarmXHistory_1.Error THEN
		MpAlarmXHistory_1.Export:= FALSE;
	ELSIF MpAlarmXHistory_1.CommandDone THEN
		MpAlarmXHistory_1.Export:= FALSE;
	END_IF

	//**********************************Porucha tlaku vzduchu*********************************************************//
	IF CasKontroly_TlakVzduchu.Q THEN
		P1_Alarmy[124]:= TRUE;
		P1_Pracovisko.STAV.Porucha_ST1:= TRUE;
		P1_Pracovisko.STAV.Porucha_ST2:= TRUE;
		P1_Pracovisko.STAV.Porucha_ST3:= TRUE;
	END_IF

	IF Safety.STAV.P1_ZonaBunky_AKTIVNA AND NOT P1_Pracovisko.IN.TlakVzduchu_OK THEN
		CasKontroly_TlakVzduchu.IN:= TRUE;
	ELSE
		CasKontroly_TlakVzduchu.IN:= FALSE;
	END_IF

	CasKontroly_TlakVzduchu.PT:= T#5s;
	CasKontroly_TlakVzduchu();

	//**********************************Porucha - kamerovy systém nieje online****************************************//
	IF CasKontroly_KAMsystem.Q THEN
		P1_Alarmy[149]:= TRUE;
		P1_Pracovisko.STAV.Porucha_ST1:= TRUE;
		P1_Pracovisko.STAV.Porucha_ST2:= TRUE;
		P1_Pracovisko.STAV.Porucha_ST3:= TRUE;
	END_IF

	IF CasKontroly_KAM3.Q THEN
		P1_Alarmy[140]:= TRUE;
		P1_Pracovisko.STAV.Porucha_ST1:= TRUE;
	END_IF

	IF CasKontroly_KAM5.Q THEN
		P1_Alarmy[141]:= TRUE;
		P1_Pracovisko.STAV.Porucha_ST1:= TRUE;
	END_IF

	IF NOT P3_Pracovisko.IN.Kamery_ControlUnit_KomOK AND P1_Pracovisko.Automat THEN
		CasKontroly_KAMsystem.IN:= TRUE;
	ELSE
		CasKontroly_KAMsystem.IN:= FALSE;
	END_IF

	IF NOT CAM3.STAV.READY AND P1_Pracovisko.Automat THEN
		CasKontroly_KAM3.IN:= TRUE;
	ELSE
		CasKontroly_KAM3.IN:= FALSE;
	END_IF

	IF NOT CAM5.STAV.READY AND P1_Pracovisko.Automat THEN
		CasKontroly_KAM5.IN:= TRUE;
	ELSE
		CasKontroly_KAM5.IN:= FALSE;
	END_IF

	CasKontroly_KAMsystem.PT:= T#2s;
	CasKontroly_KAMsystem();
	CasKontroly_KAM3.PT:= T#2s;
	CasKontroly_KAM3();
	CasKontroly_KAM5.PT:= T#2s;
	CasKontroly_KAM5();

	//**********************************Porucha - IO moduly niesu online**************************************************//
	IF CasKontroly_Moduly.Q THEN
		P1_Alarmy[125]:= TRUE;
		P1_Pracovisko.STAV.Porucha_ST1:= TRUE;
		P1_Pracovisko.STAV.Porucha_ST2:= TRUE;
		P1_Pracovisko.STAV.Porucha_ST3:= TRUE;
	END_IF

	IF Safety.STAV.P1_ZonaBunky_AKTIVNA AND (NOT P1_Pracovisko.IN.ModulFesto_IO_KomOK OR NOT P1_Pracovisko.IN.ModulWeidmuller_IO_KomOK) THEN
		CasKontroly_Moduly.IN:= TRUE;
	ELSE
		CasKontroly_Moduly.IN:= FALSE;
	END_IF

	CasKontroly_Moduly.PT:= T#2s;
	CasKontroly_Moduly();

	//********************************Porucha - ventilového terminálu**********************************************//
	IF CasKontroly_VentTerminalov.Q THEN
		P1_Alarmy[134]:= TRUE;
		P1_Pracovisko.STAV.Porucha_ST1:= TRUE;
		P1_Pracovisko.STAV.Porucha_ST2:= TRUE;
		P1_Pracovisko.STAV.Porucha_ST3:= TRUE;
	END_IF

	IF Safety.STAV.P1_ZonaBunky_AKTIVNA AND NOT P1_Pracovisko.IN.VentilovyTerminal_KomOK THEN
		CasKontroly_VentTerminalov.IN:= TRUE;
	ELSE
		CasKontroly_VentTerminalov.IN:= FALSE;
	END_IF

	CasKontroly_VentTerminalov.PT:= T#2s;
	CasKontroly_VentTerminalov();

	//********************************Porucha - skrutkovacky niesu online**********************************************//
	IF CasKontroly_Skrutkovacky.Q THEN
		IF NOT P1_Pracovisko.IN.Skrutkovacka_K30_KomOK THEN
			P1_Alarmy[136]:= TRUE;
			P1_Pracovisko.STAV.Porucha_ST2:= TRUE;
		END_IF
		IF NOT P1_Pracovisko.IN.Skrutkovacka_M5_KomOK THEN
			P1_Alarmy[137]:= TRUE;
			P1_Pracovisko.STAV.Porucha_ST2:= TRUE;
		END_IF
		IF NOT P1_Pracovisko.IN.Skrutkovacka_M4_KomOK THEN
			P1_Alarmy[138]:= TRUE;
			P1_Pracovisko.STAV.Porucha_ST2:= TRUE;
		END_IF
	END_IF

	IF Safety.STAV.P1_ZonaBunky_AKTIVNA AND (NOT P1_Pracovisko.IN.Skrutkovacka_K30_KomOK OR NOT P1_Pracovisko.IN.Skrutkovacka_M4_KomOK OR NOT P1_Pracovisko.IN.Skrutkovacka_M5_KomOK) THEN
		CasKontroly_Skrutkovacky.IN:= TRUE;
	ELSE
		CasKontroly_Skrutkovacky.IN:= FALSE;
	END_IF

	CasKontroly_Skrutkovacky.PT:= T#2s;
	CasKontroly_Skrutkovacky();

	//*********************************Porucha - robot nieje online************************************************//
	IF CasKontroly_Robota.Q THEN
		P1_Alarmy[123]:= TRUE;
		P1_Pracovisko.STAV.Porucha_ST2:= TRUE;
	END_IF

	IF Safety.STAV.P1_ZonaBunky_AKTIVNA AND NOT P1_Pracovisko.IN.Robot_KomOK THEN
		CasKontroly_Robota.IN:= TRUE;
	ELSE
		CasKontroly_Robota.IN:= FALSE;
	END_IF

	CasKontroly_Robota.PT:= T#2s;
	CasKontroly_Robota();

	//********************Pracovisko 1 - Porucha ochrannej bariéry výťahu****************************************//

	IF P1_Vytah.Automat AND NOT Safety.STAV.P1_Vytah_Bariera_AKTIVNA AND NOT Safety.STAV.P1_Vytah_Muting_AKTIVNY THEN
		P1_Alarmy[101]:= TRUE;
		P1_Pracovisko.STAV.Porucha_ST1:= TRUE;
	END_IF

	//*********************Pracovisko 1 - Porucha serva zdvihu vytahu***************//
	IF CasPoruchyServaVytahu.Q THEN
		P1_Alarmy[110]:= TRUE;
		P1_Pracovisko.STAV.Porucha_ST1:= TRUE;
	END_IF

	IF P1_Vytah.Automat AND P1_Vytah.ServoZdvihuVytahu.Status.Error THEN
		CasPoruchyServaVytahu.IN:= TRUE;
	ELSE
		CasPoruchyServaVytahu.IN:= FALSE;
	END_IF

	CasPoruchyServaVytahu.PT:= T#2s;
	CasPoruchyServaVytahu();

	//*********************Pracovisko 1 - Porucha serva manipulatora šrobovania os X***************//
	IF CasPoruchyServaSrobovaniaOsX.Q THEN
		P1_Alarmy[117]:= TRUE;
		P1_Pracovisko.STAV.Porucha_ST2:= TRUE;
	END_IF

	IF Safety.STAV.P1_ZonaBunky_AKTIVNA AND P1_Srobovanie.ServoManipulOsX.Status.Error THEN
		CasPoruchyServaSrobovaniaOsX.IN:= TRUE;
	ELSE
		CasPoruchyServaSrobovaniaOsX.IN:= FALSE;
	END_IF

	CasPoruchyServaSrobovaniaOsX.PT:= T#2s;
	CasPoruchyServaSrobovaniaOsX();

	//*********************Pracovisko 1 - Porucha serva manipulatora šrobovania os Y***************//
	IF CasPoruchyServaSrobovaniaOsY.Q THEN
		P1_Alarmy[118]:= TRUE;
		P1_Pracovisko.STAV.Porucha_ST2:= TRUE;
	END_IF

	IF Safety.STAV.P1_ZonaBunky_AKTIVNA AND P1_Srobovanie.ServoManipulOsY.Status.Error THEN
		CasPoruchyServaSrobovaniaOsY.IN:= TRUE;
	ELSE
		CasPoruchyServaSrobovaniaOsY.IN:= FALSE;
	END_IF

	CasPoruchyServaSrobovaniaOsY.PT:= T#2s;
	CasPoruchyServaSrobovaniaOsY();

	//*********************Pracovisko 1 - Porucha serva manipulatora šrobovania os Z M4***************//
	IF CasPoruchyServaSrobovaniaOsZ_M4.Q THEN
		P1_Alarmy[126]:= TRUE;
		P1_Pracovisko.STAV.Porucha_ST2:= TRUE;
	END_IF

	IF Safety.STAV.P1_ZonaBunky_AKTIVNA AND P1_Srobovanie.ServoManipulOsZ_M4.Status.Error THEN
		CasPoruchyServaSrobovaniaOsZ_M4.IN:= TRUE;
	ELSE
		CasPoruchyServaSrobovaniaOsZ_M4.IN:= FALSE;
	END_IF

	CasPoruchyServaSrobovaniaOsZ_M4.PT:= T#2s;
	CasPoruchyServaSrobovaniaOsZ_M4();

	//*********************Pracovisko 1 - Porucha serva manipulatora šrobovania os Z M5***************//
	IF CasPoruchyServaSrobovaniaOsZ_M5.Q THEN
		P1_Alarmy[127]:= TRUE;
		P1_Pracovisko.STAV.Porucha_ST2:= TRUE;
	END_IF

	IF Safety.STAV.P1_ZonaBunky_AKTIVNA AND P1_Srobovanie.ServoManipulOsZ_M5.Status.Error THEN
		CasPoruchyServaSrobovaniaOsZ_M5.IN:= TRUE;
	ELSE
		CasPoruchyServaSrobovaniaOsZ_M5.IN:= FALSE;
	END_IF

	CasPoruchyServaSrobovaniaOsZ_M5.PT:= T#2s;
	CasPoruchyServaSrobovaniaOsZ_M5();

	//********************Pracovisko 1 - Porucha skrutkovacieho setu M4******************************//
	IF P1_Srobovanie.Automat AND P1_Srobovanie.SkrutSet_M4.STAV.ERROR THEN
		P1_Alarmy[128]:= TRUE;
		P1_Pracovisko.STAV.Porucha_ST2:= TRUE;
	END_IF

	//********************Pracovisko 1 - Porucha skrutkovacieho setu M5******************************//
	IF P1_Srobovanie.Automat AND P1_Srobovanie.SkrutSet_M4.STAV.ERROR THEN
		P1_Alarmy[129]:= TRUE;
		P1_Pracovisko.STAV.Porucha_ST2:= TRUE;
	END_IF

	//****************************Pracovisko 1 - porucha vrchného dopravníka**********************************//
	IF NOT P1_Dopravniky.IN.TeplotaMotoraDopravBunky_OK AND P1_Pracovisko.STAV.Automat THEN
		P1_Alarmy[152]:= TRUE;
		P1_Pracovisko.STAV.Porucha_ST2:= TRUE;
		P1_Pracovisko.STAV.Porucha_ST3:= TRUE;
	END_IF

	//*****************************Pracovisko 1 - porucha spodného dopravníka************************************//
	IF NOT P1_Dopravniky.IN.TeplotaMotoraVratnehoDoprav_OK AND P1_Pracovisko.STAV.Automat THEN
		P1_Alarmy[153]:= TRUE;
	END_IF

	//******************************Pracovisko 1 - narušenie vstupnej bariery***********************************//
	IF CasKontrolyVstupBariery.Q THEN
		P1_Alarmy[154]:= TRUE;
		P1_Pracovisko.STAV.Porucha_ST2:= TRUE;
		P1_Pracovisko.STAV.Porucha_ST3:= TRUE;
	END_IF

	CasKontrolyVstupBariery.IN:= NOT Safety.STAV.P1_VstupBunky_VstupBar_AKTIVNA AND NOT Safety.STAV.P1_VstupBunky_VystupBar_AKTIVNA AND P1_Pracovisko.STAV.Automat;
	CasKontrolyVstupBariery.PT:= T#2s;
    CasKontrolyVstupBariery();

	//******************************Pracovisko 1 - narušenie výstupnej bariery***********************************//
	IF CasKontrolyVystupBariery.Q THEN
		P1_Alarmy[130]:= TRUE;
		P1_Pracovisko.STAV.Porucha_ST2:= TRUE;
		P1_Pracovisko.STAV.Porucha_ST3:= TRUE;
	END_IF

	CasKontrolyVystupBariery.IN:= NOT Safety.STAV.P1_VystupBunky_VstupBar_AKTIVNA AND NOT Safety.STAV.P1_VystupBunky_VystupBar_AKTIVNA AND P1_Pracovisko.STAV.Automat;
	CasKontrolyVystupBariery.PT:= T#2s;
	CasKontrolyVystupBariery();

	//******************************Výťah - porucha dopravníka**************************************************//
	IF NOT P1_Vytah.IN.TeplotaMotoraDopravVytahu_OK AND P1_Vytah.Automat THEN
		P1_Alarmy[155]:= TRUE;
		P1_Pracovisko.STAV.Porucha_ST1:= TRUE;
	END_IF

	//******************************Stlačenie tlačítok CS*******************************************************//
	IF EDGENEG(Safety.STAV.P1_Panel_TlacitkoCS_ODBLOK) THEN
		P1_Alarmy[156]:= TRUE;
	END_IF

	IF EDGENEG(Safety.STAV.P1_Rozvadzac_TlacitkoCS_ODBLOK) THEN
		P1_Alarmy[157]:= TRUE;
	END_IF

	IF EDGENEG(Safety.STAV.P1_Robot_TlacitkoCS_ODBLOK) THEN
		P1_Alarmy[158]:= TRUE;
	END_IF

	//***************************************************Nasetovanie alarmov****************************************************//
	IF P1_Alarmy[100] THEN
		MpAlarmXSet(gAlarmXCore, 'A100');
	ELSE
		MpAlarmXReset(gAlarmXCore, 'A100');
	END_IF

	IF P1_Alarmy[101] THEN
		MpAlarmXSet(gAlarmXCore, 'A101');
	ELSE
		MpAlarmXReset(gAlarmXCore, 'A101');
	END_IF

	IF P1_Alarmy[102] THEN
		MpAlarmXSet(gAlarmXCore, 'A102');
	ELSE
		MpAlarmXReset(gAlarmXCore, 'A102');
	END_IF

	IF P1_Alarmy[103] THEN
		MpAlarmXSet(gAlarmXCore, 'A103');
	ELSE
		MpAlarmXReset(gAlarmXCore, 'A103');
	END_IF

	IF P1_Alarmy[104] THEN
		MpAlarmXSet(gAlarmXCore, 'A104');
	ELSE
		MpAlarmXReset(gAlarmXCore, 'A104');
	END_IF

	IF P1_Alarmy[105] THEN
		MpAlarmXSet(gAlarmXCore, 'A105');
	ELSE
		MpAlarmXReset(gAlarmXCore, 'A105');
	END_IF

	IF P1_Alarmy[106] THEN
		MpAlarmXSet(gAlarmXCore, 'A106');
	ELSE
		MpAlarmXReset(gAlarmXCore, 'A106');
	END_IF

	IF P1_Alarmy[107] THEN
		MpAlarmXSet(gAlarmXCore, 'A107');
	ELSE
		MpAlarmXReset(gAlarmXCore, 'A107');
	END_IF

	IF P1_Alarmy[108] THEN
		MpAlarmXSet(gAlarmXCore, 'A108');
	ELSE
		MpAlarmXReset(gAlarmXCore, 'A108');
	END_IF

	IF P1_Alarmy[109] THEN
		MpAlarmXSet(gAlarmXCore, 'A109');
	ELSE
		MpAlarmXReset(gAlarmXCore, 'A109');
	END_IF

	IF P1_Alarmy[110] THEN
		MpAlarmXSet(gAlarmXCore, 'A110');
	ELSE
		MpAlarmXReset(gAlarmXCore, 'A110');
	END_IF

	IF P1_Alarmy[111] THEN
		MpAlarmXSet(gAlarmXCore, 'A111');
	ELSE
		MpAlarmXReset(gAlarmXCore, 'A111');
	END_IF

	IF P1_Alarmy[112] THEN
		MpAlarmXSet(gAlarmXCore, 'A112');
	ELSE
		MpAlarmXReset(gAlarmXCore, 'A112');
	END_IF

	IF P1_Alarmy[113] THEN
		MpAlarmXSet(gAlarmXCore, 'A113');
	ELSE
		MpAlarmXReset(gAlarmXCore, 'A113');
	END_IF

	IF P1_Alarmy[114] THEN
		MpAlarmXSet(gAlarmXCore, 'A114');
	ELSE
		MpAlarmXReset(gAlarmXCore, 'A114');
	END_IF

	IF P1_Alarmy[115] THEN
		MpAlarmXSet(gAlarmXCore, 'A115');
	ELSE
		MpAlarmXReset(gAlarmXCore, 'A115');
	END_IF

	IF P1_Alarmy[116] THEN
		MpAlarmXSet(gAlarmXCore, 'A116');
	ELSE
		MpAlarmXReset(gAlarmXCore, 'A116');
	END_IF

	IF P1_Alarmy[117] THEN
		MpAlarmXSet(gAlarmXCore, 'A117');
	ELSE
		MpAlarmXReset(gAlarmXCore, 'A117');
	END_IF

	IF P1_Alarmy[118] THEN
		MpAlarmXSet(gAlarmXCore, 'A118');
	ELSE
		MpAlarmXReset(gAlarmXCore, 'A118');
	END_IF

	IF P1_Alarmy[119] THEN
		MpAlarmXSet(gAlarmXCore, 'A119');
	ELSE
		MpAlarmXReset(gAlarmXCore, 'A119');
	END_IF

	IF P1_Alarmy[120] THEN
		MpAlarmXSet(gAlarmXCore, 'A120');
	ELSE
		MpAlarmXReset(gAlarmXCore, 'A120');
	END_IF

	IF P1_Alarmy[121] THEN
		MpAlarmXSet(gAlarmXCore, 'A121');
	ELSE
		MpAlarmXReset(gAlarmXCore, 'A121');
	END_IF

	IF P1_Alarmy[122] THEN
		MpAlarmXSet(gAlarmXCore, 'A122');
	ELSE
		MpAlarmXReset(gAlarmXCore, 'A122');
	END_IF

	IF P1_Alarmy[123] THEN
		MpAlarmXSet(gAlarmXCore, 'A123');
	ELSE
		MpAlarmXReset(gAlarmXCore, 'A123');
	END_IF

	IF P1_Alarmy[124] THEN
		MpAlarmXSet(gAlarmXCore, 'A124');
	ELSE
		MpAlarmXReset(gAlarmXCore, 'A124');
	END_IF

	IF P1_Alarmy[125] THEN
		MpAlarmXSet(gAlarmXCore, 'A125');
	ELSE
		MpAlarmXReset(gAlarmXCore, 'A125');
	END_IF

	IF P1_Alarmy[126] THEN
		MpAlarmXSet(gAlarmXCore, 'A126');
	ELSE
		MpAlarmXReset(gAlarmXCore, 'A126');
	END_IF

	IF P1_Alarmy[127] THEN
		MpAlarmXSet(gAlarmXCore, 'A127');
	ELSE
		MpAlarmXReset(gAlarmXCore, 'A127');
	END_IF

	IF P1_Alarmy[128] THEN
		MpAlarmXSet(gAlarmXCore, 'A128');
	ELSE
		MpAlarmXReset(gAlarmXCore, 'A128');
	END_IF

	IF P1_Alarmy[129] THEN
		MpAlarmXSet(gAlarmXCore, 'A129');
	ELSE
		MpAlarmXReset(gAlarmXCore, 'A129');
	END_IF

	IF P1_Alarmy[130] THEN
		MpAlarmXSet(gAlarmXCore, 'A130');
	ELSE
		MpAlarmXReset(gAlarmXCore, 'A130');
	END_IF

	IF P1_Alarmy[131] THEN
		MpAlarmXSet(gAlarmXCore, 'A131');
	ELSE
		MpAlarmXReset(gAlarmXCore, 'A131');
	END_IF

	IF P1_Alarmy[132] THEN
		MpAlarmXSet(gAlarmXCore, 'A132');
	ELSE
		MpAlarmXReset(gAlarmXCore, 'A132');
	END_IF

	IF P1_Alarmy[133] THEN
		MpAlarmXSet(gAlarmXCore, 'A133');
	ELSE
		MpAlarmXReset(gAlarmXCore, 'A133');
	END_IF

	IF P1_Alarmy[134] THEN
		MpAlarmXSet(gAlarmXCore, 'A134');
	ELSE
		MpAlarmXReset(gAlarmXCore, 'A134');
	END_IF

	IF P1_Alarmy[135] THEN
		MpAlarmXSet(gAlarmXCore, 'A135');
	ELSE
		MpAlarmXReset(gAlarmXCore, 'A135');
	END_IF

	IF P1_Alarmy[136] THEN
		MpAlarmXSet(gAlarmXCore, 'A136');
	ELSE
		MpAlarmXReset(gAlarmXCore, 'A136');
	END_IF

	IF P1_Alarmy[137] THEN
		MpAlarmXSet(gAlarmXCore, 'A137');
	ELSE
		MpAlarmXReset(gAlarmXCore, 'A137');
	END_IF

	IF P1_Alarmy[138] THEN
		MpAlarmXSet(gAlarmXCore, 'A138');
	ELSE
		MpAlarmXReset(gAlarmXCore, 'A138');
	END_IF

	IF P1_Alarmy[139] THEN
		MpAlarmXSet(gAlarmXCore, 'A139');
	ELSE
		MpAlarmXReset(gAlarmXCore, 'A139');
	END_IF

	IF P1_Alarmy[140] THEN
		MpAlarmXSet(gAlarmXCore, 'A140');
	ELSE
		MpAlarmXReset(gAlarmXCore, 'A140');
	END_IF

	IF P1_Alarmy[141] THEN
		MpAlarmXSet(gAlarmXCore, 'A141');
	ELSE
		MpAlarmXReset(gAlarmXCore, 'A141');
	END_IF

	IF P1_Alarmy[142] THEN
		MpAlarmXSet(gAlarmXCore, 'A142');
	ELSE
		MpAlarmXReset(gAlarmXCore, 'A142');
	END_IF

	IF P1_Alarmy[143] THEN
		MpAlarmXSet(gAlarmXCore, 'A143');
	ELSE
		MpAlarmXReset(gAlarmXCore, 'A143');
	END_IF

	IF P1_Alarmy[144] THEN
		MpAlarmXSet(gAlarmXCore, 'A144');
	ELSE
		MpAlarmXReset(gAlarmXCore, 'A144');
	END_IF

	IF P1_Alarmy[145] THEN
		MpAlarmXSet(gAlarmXCore, 'A145');
	ELSE
		MpAlarmXReset(gAlarmXCore, 'A145');
	END_IF

	IF P1_Alarmy[146] THEN
		MpAlarmXSet(gAlarmXCore, 'A146');
	ELSE
		MpAlarmXReset(gAlarmXCore, 'A146');
	END_IF

	IF P1_Alarmy[147] THEN
		MpAlarmXSet(gAlarmXCore, 'A147');
	ELSE
		MpAlarmXReset(gAlarmXCore, 'A147');
	END_IF

	IF P1_Alarmy[148] THEN
		MpAlarmXSet(gAlarmXCore, 'A148');
	ELSE
		MpAlarmXReset(gAlarmXCore, 'A148');
	END_IF

	IF P1_Alarmy[149] THEN
		MpAlarmXSet(gAlarmXCore, 'A149');
	ELSE
		MpAlarmXReset(gAlarmXCore, 'A149');
	END_IF

	IF P1_Alarmy[150] THEN
		MpAlarmXSet(gAlarmXCore, 'A150');
	ELSE
		MpAlarmXReset(gAlarmXCore, 'A150');
	END_IF

	IF P1_Alarmy[151] THEN
		MpAlarmXSet(gAlarmXCore, 'A151');
	ELSE
		MpAlarmXReset(gAlarmXCore, 'A151');
	END_IF

	IF P1_Alarmy[152] THEN
		MpAlarmXSet(gAlarmXCore, 'A152');
	ELSE
		MpAlarmXReset(gAlarmXCore, 'A152');
	END_IF

	IF P1_Alarmy[153] THEN
		MpAlarmXSet(gAlarmXCore, 'A153');
	ELSE
		MpAlarmXReset(gAlarmXCore, 'A153');
	END_IF

	IF P1_Alarmy[154] THEN
		MpAlarmXSet(gAlarmXCore, 'A154');
	ELSE
		MpAlarmXReset(gAlarmXCore, 'A154');
	END_IF

	IF P1_Alarmy[155] THEN
		MpAlarmXSet(gAlarmXCore, 'A155');
	ELSE
		MpAlarmXReset(gAlarmXCore, 'A155');
	END_IF

	IF P1_Alarmy[156] THEN
		MpAlarmXSet(gAlarmXCore, 'A156');
	ELSE
		MpAlarmXReset(gAlarmXCore, 'A156');
	END_IF

	IF P1_Alarmy[157] THEN
		MpAlarmXSet(gAlarmXCore, 'A157');
	ELSE
		MpAlarmXReset(gAlarmXCore, 'A157');
	END_IF

	IF P1_Alarmy[158] THEN
		MpAlarmXSet(gAlarmXCore, 'A158');
	ELSE
		MpAlarmXReset(gAlarmXCore, 'A158');
	END_IF

	IF P1_Alarmy[159] THEN
		MpAlarmXSet(gAlarmXCore, 'A159');
	ELSE
		MpAlarmXReset(gAlarmXCore, 'A159');
	END_IF

	IF P1_Alarmy[160] THEN
		MpAlarmXSet(gAlarmXCore, 'A160');
	ELSE
		MpAlarmXReset(gAlarmXCore, 'A160');
	END_IF

	IF P1_Alarmy[161] THEN
		MpAlarmXSet(gAlarmXCore, 'A161');
	ELSE
		MpAlarmXReset(gAlarmXCore, 'A161');
	END_IF

	IF P1_Alarmy[162] THEN
		MpAlarmXSet(gAlarmXCore, 'A162');
	ELSE
		MpAlarmXReset(gAlarmXCore, 'A162');
	END_IF

	IF P1_Alarmy[163] THEN
		MpAlarmXSet(gAlarmXCore, 'A163');
	ELSE
		MpAlarmXReset(gAlarmXCore, 'A163');
	END_IF

	IF P1_Alarmy[164] THEN
		MpAlarmXSet(gAlarmXCore, 'A164');
	ELSE
		MpAlarmXReset(gAlarmXCore, 'A164');
	END_IF

	IF P1_Alarmy[165] THEN
		MpAlarmXSet(gAlarmXCore, 'A165');
	ELSE
		MpAlarmXReset(gAlarmXCore, 'A165');
	END_IF

	IF P1_Alarmy[166] THEN
		MpAlarmXSet(gAlarmXCore, 'A166');
	ELSE
		MpAlarmXReset(gAlarmXCore, 'A166');
	END_IF

	IF P1_Alarmy[167] THEN
		MpAlarmXSet(gAlarmXCore, 'A167');
	ELSE
		MpAlarmXReset(gAlarmXCore, 'A167');
	END_IF

	IF P1_Alarmy[168] THEN
		MpAlarmXSet(gAlarmXCore, 'A168');
	ELSE
		MpAlarmXReset(gAlarmXCore, 'A168');
	END_IF

	//*************************************Potvrdenie alarmov*********************************************************//
	IF P1_AlarmyVizu.PotvrdAlarmy THEN
		brsmemset(ADR(P1_Alarmy),0,SIZEOF(P1_Alarmy));
		P1_Pracovisko.STAV.Porucha_ST1:= FALSE;
		P1_Pracovisko.STAV.Porucha_ST2:= FALSE;
		P1_Pracovisko.STAV.Porucha_ST3:= FALSE;
		IF NOT P1_Vytah.Automat THEN
			P1_Vytah.ServoZdvihuVytahu.Command.ErrReset:= TRUE;
		END_IF
		IF NOT P1_Srobovanie.Automat THEN
			P1_Srobovanie.ServoManipulOsX.Command.ErrReset:= TRUE;
			P1_Srobovanie.ServoManipulOsY.Command.ErrReset:= TRUE;
			P1_Srobovanie.ServoManipulOsZ_M4.Command.ErrReset:= TRUE;
			P1_Srobovanie.ServoManipulOsZ_M5.Command.ErrReset:= TRUE;
			P1_Srobovanie.SkrutSet_M4.CMD.ResetPoruchy:= TRUE;
			P1_Srobovanie.SkrutSet_M5.CMD.ResetPoruchy:= TRUE;
		END_IF
		P1_AlarmyVizu.PotvrdAlarmy:= FALSE;
	END_IF

    END_PROGRAM

PROGRAM _EXIT
        (* Insert code here *)

        END_PROGRAM
```

#### Variables.var - Local variables
```iecst
VAR
	i : UINT;
	CasKontroly_KAMsystem : TON;
	CasKontroly_TlakVzduchu : TON;
	CasKontroly_Moduly : TON;
	CasKontroly_Robota : TON;
	CasKontroly_VentTerminalov : TON;
	CasKontroly_Skrutkovacky : TON;
	CasPoruchyServaVytahu : TON;
	CasPoruchyServaSrobovaniaOsY : TON;
	CasPoruchyServaSrobovaniaOsX : TON;
	CasResetovaniaServaZdvihuVytahu : TON;
	CasResetovaniaServaSrobovaniaOsX : TON;
	CasResetovaniaServaSrobovaniaOsY : TON;
	a : INT;
	CasKontroly_KAM3 : TON;
	CasKontroly_KAM5 : TON;
	CasKontroly_ModulyVytahu : TON;
	CasKontroly_ModulyBunky : TON;
	CasPoruchyServaSrobovaniaOsZ_M4 : TON;
	CasPoruchyServaSrobovaniaOsZ_M5 : TON;
	CasKontrolyVstupBariery : TON := (0);
	CasKontrolyVystupBariery : TON;
	TT : BOOL := 0;
END_VAR
```

### Program Logical/Alarmy/P2_Alarmy (IEC)
